// TIA Portal V20 export
FUNCTION_BLOCK "EmOverviewHomeCondition"   // FB5, LAD
// stored: MemoryReserve 100, SetENOAutomatically false
   VAR
      statMaxPageCount : Array[0..13] of Int;
      statPulse { ExternalAccessible := 'False'; ExternalVisible := 'False'; ExternalWritable := 'False'} : Array[0..199] of Bool;
      statLampOff { ExternalAccessible := 'False'; ExternalVisible := 'False'; ExternalWritable := 'False'} : Array[0..13] of Bool;
      statLampControl { ExternalAccessible := 'False'; ExternalVisible := 'False'; ExternalWritable := 'False'} : Bool;
   END_VAR
   VAR CONSTANT
      TRUE : Bool := TRUE;
      FALSE : Bool := FALSE;
   END_VAR
   VAR_TEMP   // added for the SCL form of the ladder/FBD networks
      _w1 : Bool;
      _w2 : Bool;
   END_VAR
BEGIN

REGION Network 1: Lamp Control
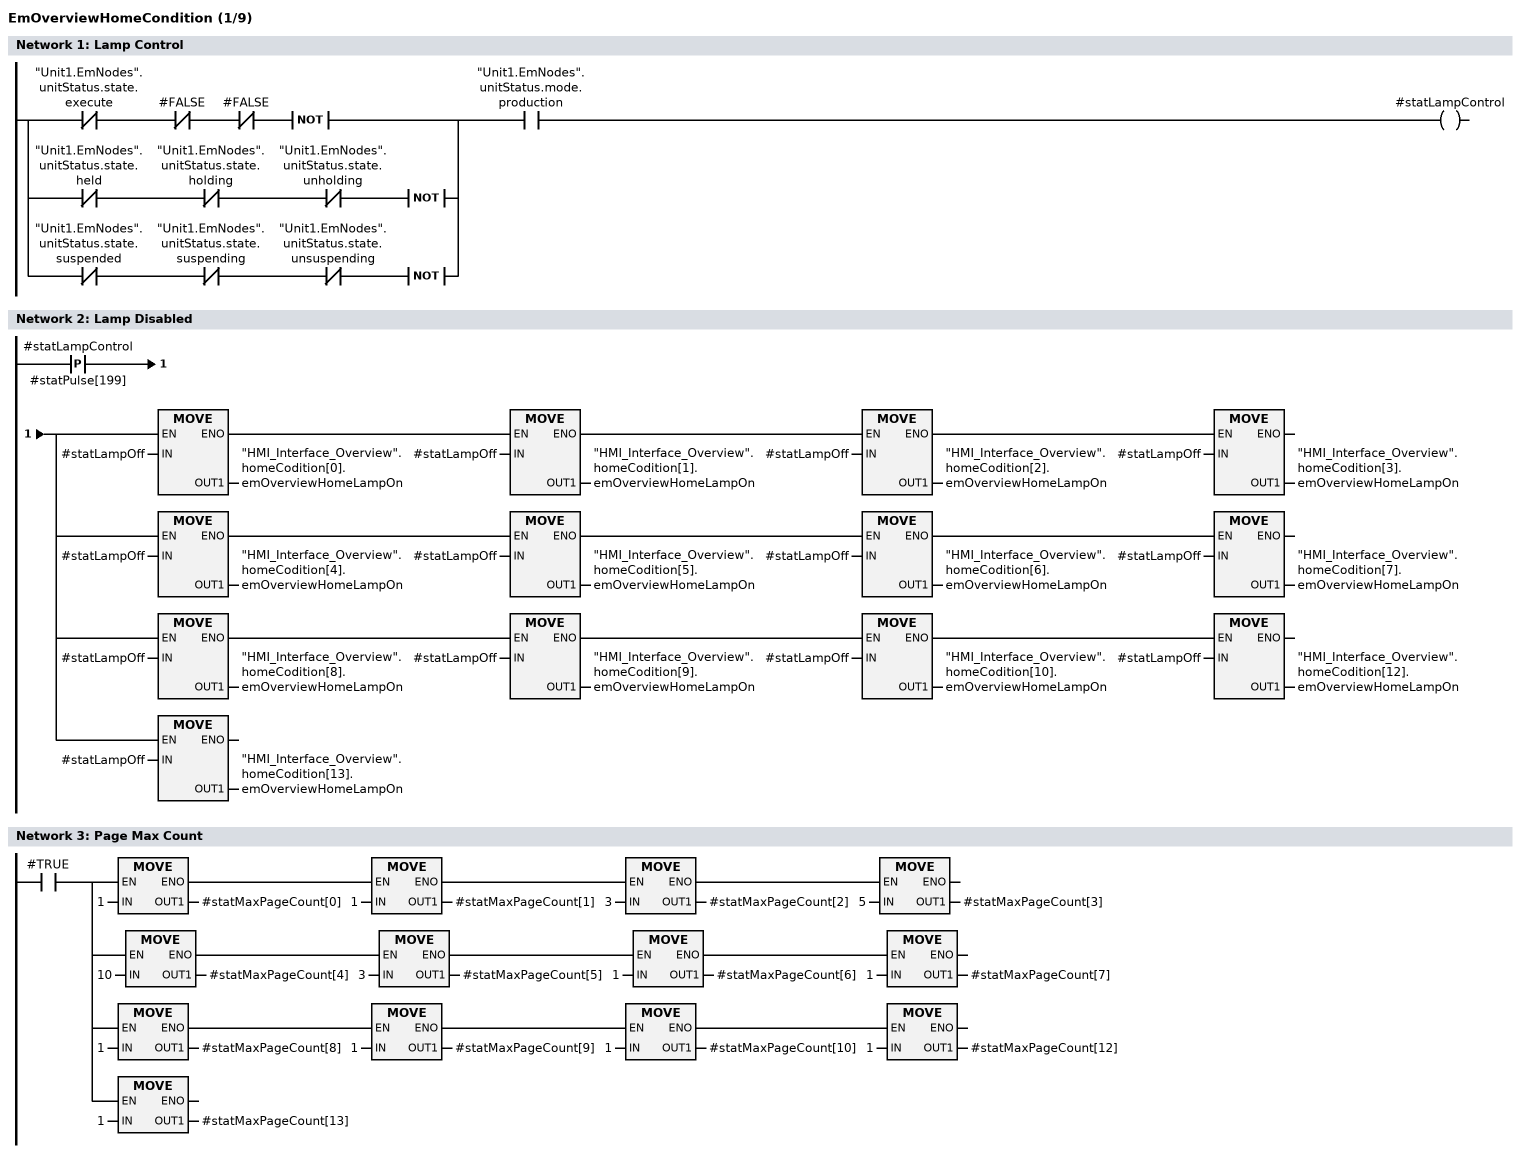
   RUNG wire#powerrail
      I_Contact( "Unit1.EmNodes".unitStatus.state.execute )
      I_Contact( #FALSE )
      I_Contact( #FALSE )
      Not()
      wire#w1
      Contact( "Unit1.EmNodes".unitStatus.mode.production )
      Coil( #statLampControl )
   END_RUNG
   RUNG wire#powerrail
      I_Contact( "Unit1.EmNodes".unitStatus.state.held )
      I_Contact( "Unit1.EmNodes".unitStatus.state.holding )
      I_Contact( "Unit1.EmNodes".unitStatus.state.unholding )
      Not()
   END_RUNG wire#w1
   RUNG wire#powerrail
      I_Contact( "Unit1.EmNodes".unitStatus.state.suspended )
      I_Contact( "Unit1.EmNodes".unitStatus.state.suspending )
      I_Contact( "Unit1.EmNodes".unitStatus.state.unsuspending )
      Not()
   END_RUNG wire#w1
   // the same network as SCL:
   #statLampControl := (NOT (NOT "Unit1.EmNodes".unitStatus.state.execute AND NOT #FALSE AND NOT #FALSE) OR NOT (NOT "Unit1.EmNodes".unitStatus.state.held AND NOT "Unit1.EmNodes".unitStatus.state.holding AND NOT "Unit1.EmNodes".unitStatus.state.unholding) OR NOT (NOT "Unit1.EmNodes".unitStatus.state.suspended AND NOT "Unit1.EmNodes".unitStatus.state.suspending AND NOT "Unit1.EmNodes".unitStatus.state.unsuspending)) AND "Unit1.EmNodes".unitStatus.mode.production;
END_REGION

REGION Network 2: Lamp Disabled
   RUNG wire#powerrail
      P_Contact(operand := #statLampControl, bit := #statPulse[199])
      wire#w1
      Move(in := #statLampOff, out1 => "HMI_Interface_Overview".homeCodition[0].emOverviewHomeLampOn)
      Move(in := #statLampOff, out1 => "HMI_Interface_Overview".homeCodition[1].emOverviewHomeLampOn)
      Move(in := #statLampOff, out1 => "HMI_Interface_Overview".homeCodition[2].emOverviewHomeLampOn)
      Move(in := #statLampOff, out1 => "HMI_Interface_Overview".homeCodition[3].emOverviewHomeLampOn)
   END_RUNG
   RUNG wire#w1
      Move(in := #statLampOff, out1 => "HMI_Interface_Overview".homeCodition[4].emOverviewHomeLampOn)
      Move(in := #statLampOff, out1 => "HMI_Interface_Overview".homeCodition[5].emOverviewHomeLampOn)
      Move(in := #statLampOff, out1 => "HMI_Interface_Overview".homeCodition[6].emOverviewHomeLampOn)
      Move(in := #statLampOff, out1 => "HMI_Interface_Overview".homeCodition[7].emOverviewHomeLampOn)
   END_RUNG
   RUNG wire#w1
      Move(in := #statLampOff, out1 => "HMI_Interface_Overview".homeCodition[8].emOverviewHomeLampOn)
      Move(in := #statLampOff, out1 => "HMI_Interface_Overview".homeCodition[9].emOverviewHomeLampOn)
      Move(in := #statLampOff, out1 => "HMI_Interface_Overview".homeCodition[10].emOverviewHomeLampOn)
      Move(in := #statLampOff, out1 => "HMI_Interface_Overview".homeCodition[12].emOverviewHomeLampOn)
   END_RUNG
   RUNG wire#w1
      Move(in := #statLampOff, out1 => "HMI_Interface_Overview".homeCodition[13].emOverviewHomeLampOn)
   END_RUNG
   // the same network as SCL:
   #_w1 := #statLampControl AND NOT #statPulse[199];   // rising edge of #statLampControl
   #statPulse[199] := #statLampControl;
   IF #_w1 THEN
       "HMI_Interface_Overview".homeCodition[0].emOverviewHomeLampOn := #statLampOff;
       "HMI_Interface_Overview".homeCodition[1].emOverviewHomeLampOn := #statLampOff;
       "HMI_Interface_Overview".homeCodition[2].emOverviewHomeLampOn := #statLampOff;
       "HMI_Interface_Overview".homeCodition[3].emOverviewHomeLampOn := #statLampOff;
       "HMI_Interface_Overview".homeCodition[4].emOverviewHomeLampOn := #statLampOff;
       "HMI_Interface_Overview".homeCodition[5].emOverviewHomeLampOn := #statLampOff;
       "HMI_Interface_Overview".homeCodition[6].emOverviewHomeLampOn := #statLampOff;
       "HMI_Interface_Overview".homeCodition[7].emOverviewHomeLampOn := #statLampOff;
       "HMI_Interface_Overview".homeCodition[8].emOverviewHomeLampOn := #statLampOff;
       "HMI_Interface_Overview".homeCodition[9].emOverviewHomeLampOn := #statLampOff;
       "HMI_Interface_Overview".homeCodition[10].emOverviewHomeLampOn := #statLampOff;
       "HMI_Interface_Overview".homeCodition[12].emOverviewHomeLampOn := #statLampOff;
       "HMI_Interface_Overview".homeCodition[13].emOverviewHomeLampOn := #statLampOff;
   END_IF;
END_REGION

REGION Network 3: Page Max Count
   RUNG wire#powerrail
      Contact( #TRUE )
      wire#w1
      Move(in := 1, out1 => #statMaxPageCount[0])
      Move(in := 1, out1 => #statMaxPageCount[1])
      Move(in := 3, out1 => #statMaxPageCount[2])
      Move(in := 5, out1 => #statMaxPageCount[3])
   END_RUNG
   RUNG wire#w1
      Move(in := 10, out1 => #statMaxPageCount[4])
      Move(in := 3, out1 => #statMaxPageCount[5])
      Move(in := 1, out1 => #statMaxPageCount[6])
      Move(in := 1, out1 => #statMaxPageCount[7])
   END_RUNG
   RUNG wire#w1
      Move(in := 1, out1 => #statMaxPageCount[8])
      Move(in := 1, out1 => #statMaxPageCount[9])
      Move(in := 1, out1 => #statMaxPageCount[10])
      Move(in := 1, out1 => #statMaxPageCount[12])
   END_RUNG
   RUNG wire#w1
      Move(in := 1, out1 => #statMaxPageCount[13])
   END_RUNG
   // the same network as SCL:
   IF #TRUE THEN
       #statMaxPageCount[0] := 1;
       #statMaxPageCount[1] := 1;
       #statMaxPageCount[2] := 3;
       #statMaxPageCount[3] := 5;
       #statMaxPageCount[4] := 10;
       #statMaxPageCount[5] := 3;
       #statMaxPageCount[6] := 1;
       #statMaxPageCount[7] := 1;
       #statMaxPageCount[8] := 1;
       #statMaxPageCount[9] := 1;
       #statMaxPageCount[10] := 1;
       #statMaxPageCount[12] := 1;
       #statMaxPageCount[13] := 1;
   END_IF;
END_REGION

REGION Network 4: Em 0 Page Index Control
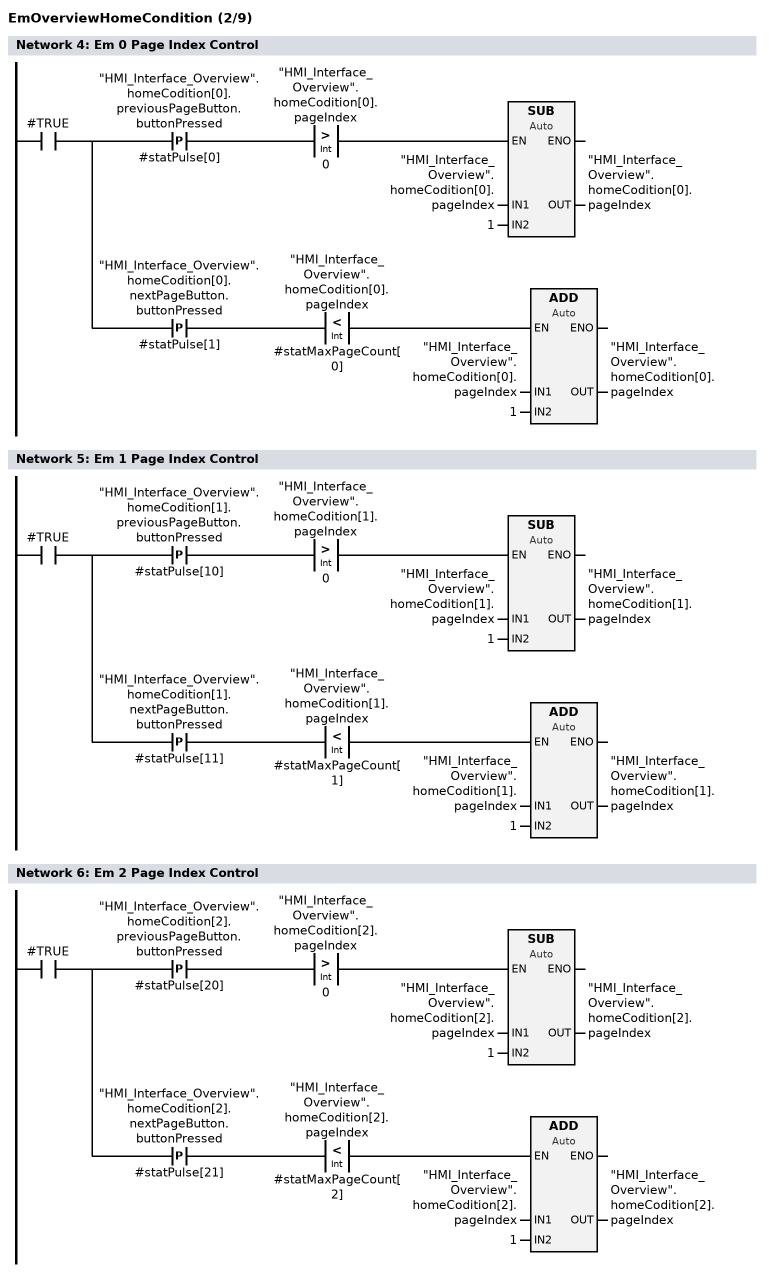
   RUNG wire#powerrail
      Contact( #TRUE )
      wire#w1
      P_Contact(operand := "HMI_Interface_Overview".homeCodition[0].previousPageButton.buttonPressed, bit := #statPulse[0])
      { S7_Templates := "SrcType := Int" } GT_Contact(in1 := "HMI_Interface_Overview".homeCodition[0].pageIndex, in2 := 0)
      Sub(in1 := "HMI_Interface_Overview".homeCodition[0].pageIndex, in2 := 1, out => "HMI_Interface_Overview".homeCodition[0].pageIndex)
   END_RUNG
   RUNG wire#w1
      P_Contact(operand := "HMI_Interface_Overview".homeCodition[0].nextPageButton.buttonPressed, bit := #statPulse[1])
      { S7_Templates := "SrcType := Int" } LT_Contact(in1 := "HMI_Interface_Overview".homeCodition[0].pageIndex, in2 := #statMaxPageCount[0])
      Add(in1 := "HMI_Interface_Overview".homeCodition[0].pageIndex, in2 := 1, out => "HMI_Interface_Overview".homeCodition[0].pageIndex)
   END_RUNG
   // the same network as SCL:
   #_w1 := #TRUE AND "HMI_Interface_Overview".homeCodition[0].previousPageButton.buttonPressed AND NOT #statPulse[0];   // rising edge of "HMI_Interface_Overview".homeCodition[0].previousPageButton.buttonPressed
   #statPulse[0] := "HMI_Interface_Overview".homeCodition[0].previousPageButton.buttonPressed;
   IF #_w1 AND ("HMI_Interface_Overview".homeCodition[0].pageIndex > 0) THEN
       "HMI_Interface_Overview".homeCodition[0].pageIndex := "HMI_Interface_Overview".homeCodition[0].pageIndex - 1;
   END_IF;
   #_w2 := #TRUE AND "HMI_Interface_Overview".homeCodition[0].nextPageButton.buttonPressed AND NOT #statPulse[1];   // rising edge of "HMI_Interface_Overview".homeCodition[0].nextPageButton.buttonPressed
   #statPulse[1] := "HMI_Interface_Overview".homeCodition[0].nextPageButton.buttonPressed;
   IF #_w2 AND ("HMI_Interface_Overview".homeCodition[0].pageIndex < #statMaxPageCount[0]) THEN
       "HMI_Interface_Overview".homeCodition[0].pageIndex := "HMI_Interface_Overview".homeCodition[0].pageIndex + 1;
   END_IF;
END_REGION

REGION Network 5: Em 1 Page Index Control
   RUNG wire#powerrail
      Contact( #TRUE )
      wire#w1
      P_Contact(operand := "HMI_Interface_Overview".homeCodition[1].previousPageButton.buttonPressed, bit := #statPulse[10])
      { S7_Templates := "SrcType := Int" } GT_Contact(in1 := "HMI_Interface_Overview".homeCodition[1].pageIndex, in2 := 0)
      Sub(in1 := "HMI_Interface_Overview".homeCodition[1].pageIndex, in2 := 1, out => "HMI_Interface_Overview".homeCodition[1].pageIndex)
   END_RUNG
   RUNG wire#w1
      P_Contact(operand := "HMI_Interface_Overview".homeCodition[1].nextPageButton.buttonPressed, bit := #statPulse[11])
      { S7_Templates := "SrcType := Int" } LT_Contact(in1 := "HMI_Interface_Overview".homeCodition[1].pageIndex, in2 := #statMaxPageCount[1])
      Add(in1 := "HMI_Interface_Overview".homeCodition[1].pageIndex, in2 := 1, out => "HMI_Interface_Overview".homeCodition[1].pageIndex)
   END_RUNG
   // the same network as SCL:
   #_w1 := #TRUE AND "HMI_Interface_Overview".homeCodition[1].previousPageButton.buttonPressed AND NOT #statPulse[10];   // rising edge of "HMI_Interface_Overview".homeCodition[1].previousPageButton.buttonPressed
   #statPulse[10] := "HMI_Interface_Overview".homeCodition[1].previousPageButton.buttonPressed;
   IF #_w1 AND ("HMI_Interface_Overview".homeCodition[1].pageIndex > 0) THEN
       "HMI_Interface_Overview".homeCodition[1].pageIndex := "HMI_Interface_Overview".homeCodition[1].pageIndex - 1;
   END_IF;
   #_w2 := #TRUE AND "HMI_Interface_Overview".homeCodition[1].nextPageButton.buttonPressed AND NOT #statPulse[11];   // rising edge of "HMI_Interface_Overview".homeCodition[1].nextPageButton.buttonPressed
   #statPulse[11] := "HMI_Interface_Overview".homeCodition[1].nextPageButton.buttonPressed;
   IF #_w2 AND ("HMI_Interface_Overview".homeCodition[1].pageIndex < #statMaxPageCount[1]) THEN
       "HMI_Interface_Overview".homeCodition[1].pageIndex := "HMI_Interface_Overview".homeCodition[1].pageIndex + 1;
   END_IF;
END_REGION

REGION Network 6: Em 2 Page Index Control
   RUNG wire#powerrail
      Contact( #TRUE )
      wire#w1
      P_Contact(operand := "HMI_Interface_Overview".homeCodition[2].previousPageButton.buttonPressed, bit := #statPulse[20])
      { S7_Templates := "SrcType := Int" } GT_Contact(in1 := "HMI_Interface_Overview".homeCodition[2].pageIndex, in2 := 0)
      Sub(in1 := "HMI_Interface_Overview".homeCodition[2].pageIndex, in2 := 1, out => "HMI_Interface_Overview".homeCodition[2].pageIndex)
   END_RUNG
   RUNG wire#w1
      P_Contact(operand := "HMI_Interface_Overview".homeCodition[2].nextPageButton.buttonPressed, bit := #statPulse[21])
      { S7_Templates := "SrcType := Int" } LT_Contact(in1 := "HMI_Interface_Overview".homeCodition[2].pageIndex, in2 := #statMaxPageCount[2])
      Add(in1 := "HMI_Interface_Overview".homeCodition[2].pageIndex, in2 := 1, out => "HMI_Interface_Overview".homeCodition[2].pageIndex)
   END_RUNG
   // the same network as SCL:
   #_w1 := #TRUE AND "HMI_Interface_Overview".homeCodition[2].previousPageButton.buttonPressed AND NOT #statPulse[20];   // rising edge of "HMI_Interface_Overview".homeCodition[2].previousPageButton.buttonPressed
   #statPulse[20] := "HMI_Interface_Overview".homeCodition[2].previousPageButton.buttonPressed;
   IF #_w1 AND ("HMI_Interface_Overview".homeCodition[2].pageIndex > 0) THEN
       "HMI_Interface_Overview".homeCodition[2].pageIndex := "HMI_Interface_Overview".homeCodition[2].pageIndex - 1;
   END_IF;
   #_w2 := #TRUE AND "HMI_Interface_Overview".homeCodition[2].nextPageButton.buttonPressed AND NOT #statPulse[21];   // rising edge of "HMI_Interface_Overview".homeCodition[2].nextPageButton.buttonPressed
   #statPulse[21] := "HMI_Interface_Overview".homeCodition[2].nextPageButton.buttonPressed;
   IF #_w2 AND ("HMI_Interface_Overview".homeCodition[2].pageIndex < #statMaxPageCount[2]) THEN
       "HMI_Interface_Overview".homeCodition[2].pageIndex := "HMI_Interface_Overview".homeCodition[2].pageIndex + 1;
   END_IF;
END_REGION

REGION Network 7: Em 3 Page Index Control
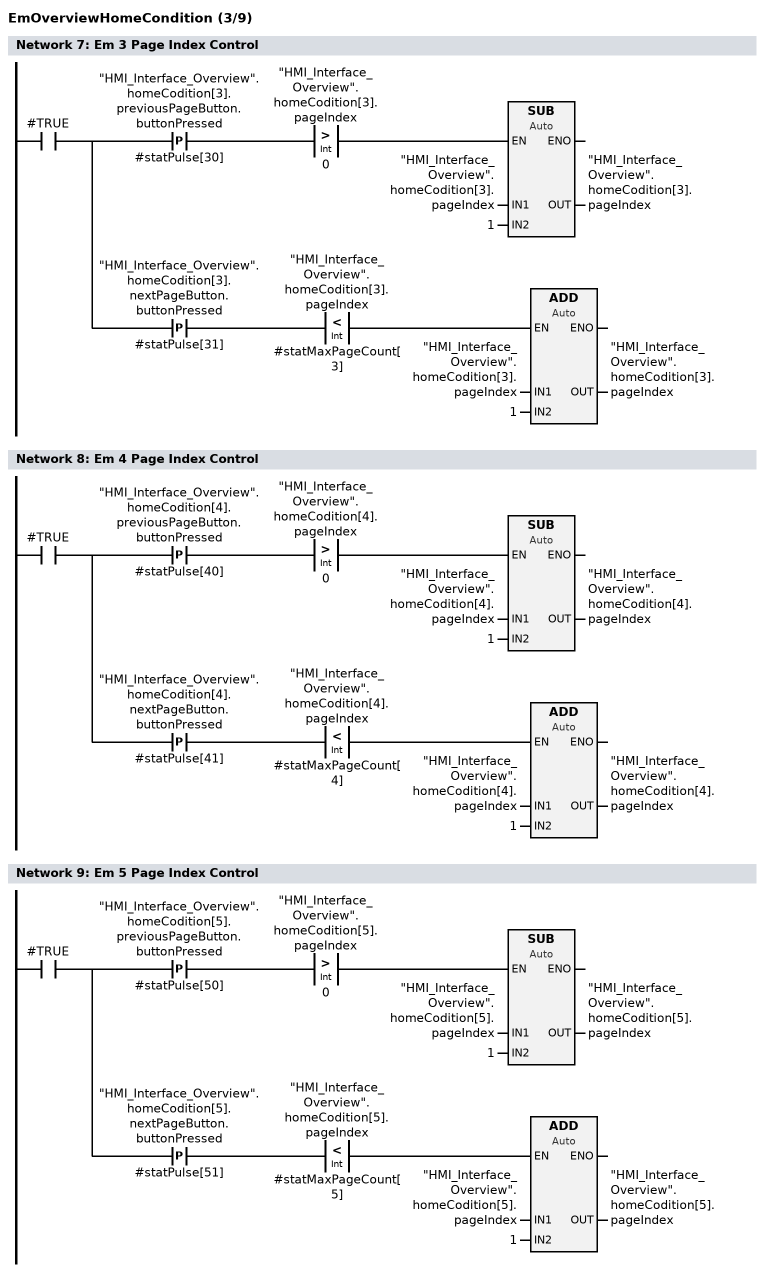
   RUNG wire#powerrail
      Contact( #TRUE )
      wire#w1
      P_Contact(operand := "HMI_Interface_Overview".homeCodition[3].previousPageButton.buttonPressed, bit := #statPulse[30])
      { S7_Templates := "SrcType := Int" } GT_Contact(in1 := "HMI_Interface_Overview".homeCodition[3].pageIndex, in2 := 0)
      Sub(in1 := "HMI_Interface_Overview".homeCodition[3].pageIndex, in2 := 1, out => "HMI_Interface_Overview".homeCodition[3].pageIndex)
   END_RUNG
   RUNG wire#w1
      P_Contact(operand := "HMI_Interface_Overview".homeCodition[3].nextPageButton.buttonPressed, bit := #statPulse[31])
      { S7_Templates := "SrcType := Int" } LT_Contact(in1 := "HMI_Interface_Overview".homeCodition[3].pageIndex, in2 := #statMaxPageCount[3])
      Add(in1 := "HMI_Interface_Overview".homeCodition[3].pageIndex, in2 := 1, out => "HMI_Interface_Overview".homeCodition[3].pageIndex)
   END_RUNG
   // the same network as SCL:
   #_w1 := #TRUE AND "HMI_Interface_Overview".homeCodition[3].previousPageButton.buttonPressed AND NOT #statPulse[30];   // rising edge of "HMI_Interface_Overview".homeCodition[3].previousPageButton.buttonPressed
   #statPulse[30] := "HMI_Interface_Overview".homeCodition[3].previousPageButton.buttonPressed;
   IF #_w1 AND ("HMI_Interface_Overview".homeCodition[3].pageIndex > 0) THEN
       "HMI_Interface_Overview".homeCodition[3].pageIndex := "HMI_Interface_Overview".homeCodition[3].pageIndex - 1;
   END_IF;
   #_w2 := #TRUE AND "HMI_Interface_Overview".homeCodition[3].nextPageButton.buttonPressed AND NOT #statPulse[31];   // rising edge of "HMI_Interface_Overview".homeCodition[3].nextPageButton.buttonPressed
   #statPulse[31] := "HMI_Interface_Overview".homeCodition[3].nextPageButton.buttonPressed;
   IF #_w2 AND ("HMI_Interface_Overview".homeCodition[3].pageIndex < #statMaxPageCount[3]) THEN
       "HMI_Interface_Overview".homeCodition[3].pageIndex := "HMI_Interface_Overview".homeCodition[3].pageIndex + 1;
   END_IF;
END_REGION

REGION Network 8: Em 4 Page Index Control
   RUNG wire#powerrail
      Contact( #TRUE )
      wire#w1
      P_Contact(operand := "HMI_Interface_Overview".homeCodition[4].previousPageButton.buttonPressed, bit := #statPulse[40])
      { S7_Templates := "SrcType := Int" } GT_Contact(in1 := "HMI_Interface_Overview".homeCodition[4].pageIndex, in2 := 0)
      Sub(in1 := "HMI_Interface_Overview".homeCodition[4].pageIndex, in2 := 1, out => "HMI_Interface_Overview".homeCodition[4].pageIndex)
   END_RUNG
   RUNG wire#w1
      P_Contact(operand := "HMI_Interface_Overview".homeCodition[4].nextPageButton.buttonPressed, bit := #statPulse[41])
      { S7_Templates := "SrcType := Int" } LT_Contact(in1 := "HMI_Interface_Overview".homeCodition[4].pageIndex, in2 := #statMaxPageCount[4])
      Add(in1 := "HMI_Interface_Overview".homeCodition[4].pageIndex, in2 := 1, out => "HMI_Interface_Overview".homeCodition[4].pageIndex)
   END_RUNG
   // the same network as SCL:
   #_w1 := #TRUE AND "HMI_Interface_Overview".homeCodition[4].previousPageButton.buttonPressed AND NOT #statPulse[40];   // rising edge of "HMI_Interface_Overview".homeCodition[4].previousPageButton.buttonPressed
   #statPulse[40] := "HMI_Interface_Overview".homeCodition[4].previousPageButton.buttonPressed;
   IF #_w1 AND ("HMI_Interface_Overview".homeCodition[4].pageIndex > 0) THEN
       "HMI_Interface_Overview".homeCodition[4].pageIndex := "HMI_Interface_Overview".homeCodition[4].pageIndex - 1;
   END_IF;
   #_w2 := #TRUE AND "HMI_Interface_Overview".homeCodition[4].nextPageButton.buttonPressed AND NOT #statPulse[41];   // rising edge of "HMI_Interface_Overview".homeCodition[4].nextPageButton.buttonPressed
   #statPulse[41] := "HMI_Interface_Overview".homeCodition[4].nextPageButton.buttonPressed;
   IF #_w2 AND ("HMI_Interface_Overview".homeCodition[4].pageIndex < #statMaxPageCount[4]) THEN
       "HMI_Interface_Overview".homeCodition[4].pageIndex := "HMI_Interface_Overview".homeCodition[4].pageIndex + 1;
   END_IF;
END_REGION

REGION Network 9: Em 5 Page Index Control
   RUNG wire#powerrail
      Contact( #TRUE )
      wire#w1
      P_Contact(operand := "HMI_Interface_Overview".homeCodition[5].previousPageButton.buttonPressed, bit := #statPulse[50])
      { S7_Templates := "SrcType := Int" } GT_Contact(in1 := "HMI_Interface_Overview".homeCodition[5].pageIndex, in2 := 0)
      Sub(in1 := "HMI_Interface_Overview".homeCodition[5].pageIndex, in2 := 1, out => "HMI_Interface_Overview".homeCodition[5].pageIndex)
   END_RUNG
   RUNG wire#w1
      P_Contact(operand := "HMI_Interface_Overview".homeCodition[5].nextPageButton.buttonPressed, bit := #statPulse[51])
      { S7_Templates := "SrcType := Int" } LT_Contact(in1 := "HMI_Interface_Overview".homeCodition[5].pageIndex, in2 := #statMaxPageCount[5])
      Add(in1 := "HMI_Interface_Overview".homeCodition[5].pageIndex, in2 := 1, out => "HMI_Interface_Overview".homeCodition[5].pageIndex)
   END_RUNG
   // the same network as SCL:
   #_w1 := #TRUE AND "HMI_Interface_Overview".homeCodition[5].previousPageButton.buttonPressed AND NOT #statPulse[50];   // rising edge of "HMI_Interface_Overview".homeCodition[5].previousPageButton.buttonPressed
   #statPulse[50] := "HMI_Interface_Overview".homeCodition[5].previousPageButton.buttonPressed;
   IF #_w1 AND ("HMI_Interface_Overview".homeCodition[5].pageIndex > 0) THEN
       "HMI_Interface_Overview".homeCodition[5].pageIndex := "HMI_Interface_Overview".homeCodition[5].pageIndex - 1;
   END_IF;
   #_w2 := #TRUE AND "HMI_Interface_Overview".homeCodition[5].nextPageButton.buttonPressed AND NOT #statPulse[51];   // rising edge of "HMI_Interface_Overview".homeCodition[5].nextPageButton.buttonPressed
   #statPulse[51] := "HMI_Interface_Overview".homeCodition[5].nextPageButton.buttonPressed;
   IF #_w2 AND ("HMI_Interface_Overview".homeCodition[5].pageIndex < #statMaxPageCount[5]) THEN
       "HMI_Interface_Overview".homeCodition[5].pageIndex := "HMI_Interface_Overview".homeCodition[5].pageIndex + 1;
   END_IF;
END_REGION

REGION Network 10: Em 6 Page Index Control
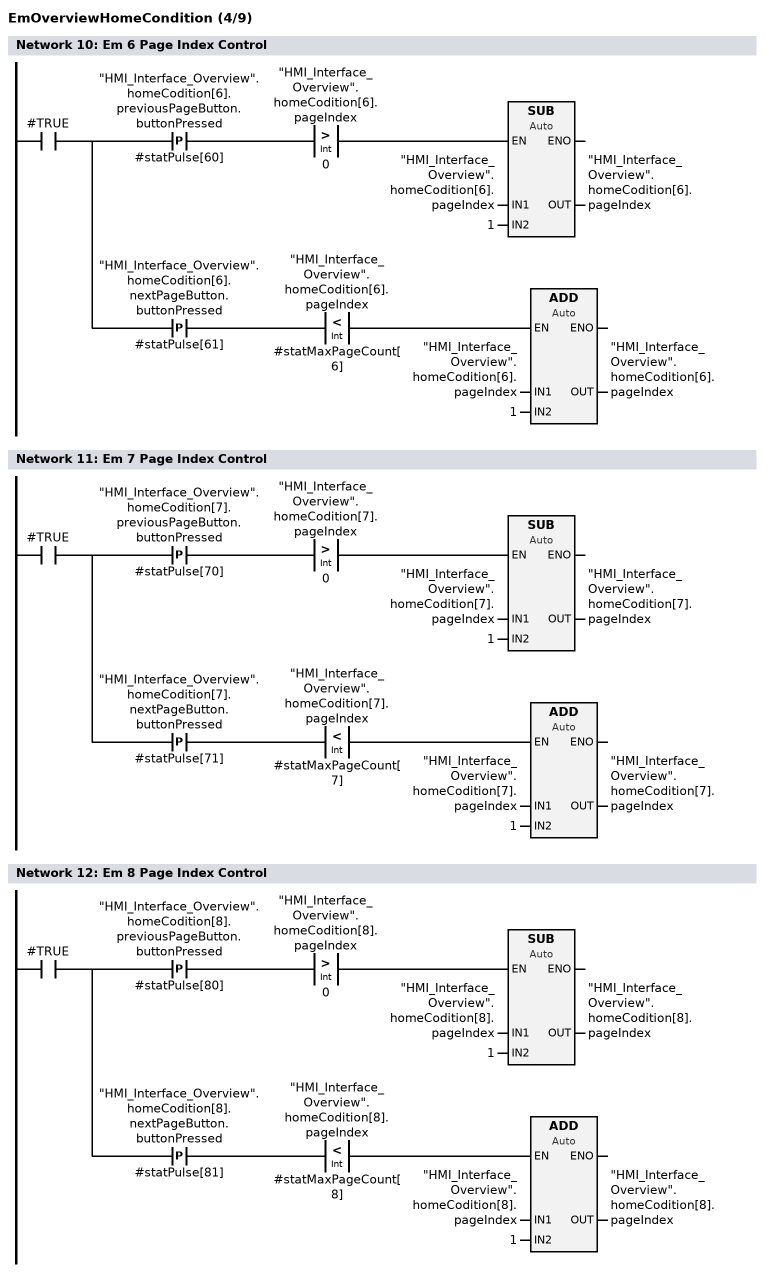
   RUNG wire#powerrail
      Contact( #TRUE )
      wire#w1
      P_Contact(operand := "HMI_Interface_Overview".homeCodition[6].previousPageButton.buttonPressed, bit := #statPulse[60])
      { S7_Templates := "SrcType := Int" } GT_Contact(in1 := "HMI_Interface_Overview".homeCodition[6].pageIndex, in2 := 0)
      Sub(in1 := "HMI_Interface_Overview".homeCodition[6].pageIndex, in2 := 1, out => "HMI_Interface_Overview".homeCodition[6].pageIndex)
   END_RUNG
   RUNG wire#w1
      P_Contact(operand := "HMI_Interface_Overview".homeCodition[6].nextPageButton.buttonPressed, bit := #statPulse[61])
      { S7_Templates := "SrcType := Int" } LT_Contact(in1 := "HMI_Interface_Overview".homeCodition[6].pageIndex, in2 := #statMaxPageCount[6])
      Add(in1 := "HMI_Interface_Overview".homeCodition[6].pageIndex, in2 := 1, out => "HMI_Interface_Overview".homeCodition[6].pageIndex)
   END_RUNG
   // the same network as SCL:
   #_w1 := #TRUE AND "HMI_Interface_Overview".homeCodition[6].previousPageButton.buttonPressed AND NOT #statPulse[60];   // rising edge of "HMI_Interface_Overview".homeCodition[6].previousPageButton.buttonPressed
   #statPulse[60] := "HMI_Interface_Overview".homeCodition[6].previousPageButton.buttonPressed;
   IF #_w1 AND ("HMI_Interface_Overview".homeCodition[6].pageIndex > 0) THEN
       "HMI_Interface_Overview".homeCodition[6].pageIndex := "HMI_Interface_Overview".homeCodition[6].pageIndex - 1;
   END_IF;
   #_w2 := #TRUE AND "HMI_Interface_Overview".homeCodition[6].nextPageButton.buttonPressed AND NOT #statPulse[61];   // rising edge of "HMI_Interface_Overview".homeCodition[6].nextPageButton.buttonPressed
   #statPulse[61] := "HMI_Interface_Overview".homeCodition[6].nextPageButton.buttonPressed;
   IF #_w2 AND ("HMI_Interface_Overview".homeCodition[6].pageIndex < #statMaxPageCount[6]) THEN
       "HMI_Interface_Overview".homeCodition[6].pageIndex := "HMI_Interface_Overview".homeCodition[6].pageIndex + 1;
   END_IF;
END_REGION

REGION Network 11: Em 7 Page Index Control
   RUNG wire#powerrail
      Contact( #TRUE )
      wire#w1
      P_Contact(operand := "HMI_Interface_Overview".homeCodition[7].previousPageButton.buttonPressed, bit := #statPulse[70])
      { S7_Templates := "SrcType := Int" } GT_Contact(in1 := "HMI_Interface_Overview".homeCodition[7].pageIndex, in2 := 0)
      Sub(in1 := "HMI_Interface_Overview".homeCodition[7].pageIndex, in2 := 1, out => "HMI_Interface_Overview".homeCodition[7].pageIndex)
   END_RUNG
   RUNG wire#w1
      P_Contact(operand := "HMI_Interface_Overview".homeCodition[7].nextPageButton.buttonPressed, bit := #statPulse[71])
      { S7_Templates := "SrcType := Int" } LT_Contact(in1 := "HMI_Interface_Overview".homeCodition[7].pageIndex, in2 := #statMaxPageCount[7])
      Add(in1 := "HMI_Interface_Overview".homeCodition[7].pageIndex, in2 := 1, out => "HMI_Interface_Overview".homeCodition[7].pageIndex)
   END_RUNG
   // the same network as SCL:
   #_w1 := #TRUE AND "HMI_Interface_Overview".homeCodition[7].previousPageButton.buttonPressed AND NOT #statPulse[70];   // rising edge of "HMI_Interface_Overview".homeCodition[7].previousPageButton.buttonPressed
   #statPulse[70] := "HMI_Interface_Overview".homeCodition[7].previousPageButton.buttonPressed;
   IF #_w1 AND ("HMI_Interface_Overview".homeCodition[7].pageIndex > 0) THEN
       "HMI_Interface_Overview".homeCodition[7].pageIndex := "HMI_Interface_Overview".homeCodition[7].pageIndex - 1;
   END_IF;
   #_w2 := #TRUE AND "HMI_Interface_Overview".homeCodition[7].nextPageButton.buttonPressed AND NOT #statPulse[71];   // rising edge of "HMI_Interface_Overview".homeCodition[7].nextPageButton.buttonPressed
   #statPulse[71] := "HMI_Interface_Overview".homeCodition[7].nextPageButton.buttonPressed;
   IF #_w2 AND ("HMI_Interface_Overview".homeCodition[7].pageIndex < #statMaxPageCount[7]) THEN
       "HMI_Interface_Overview".homeCodition[7].pageIndex := "HMI_Interface_Overview".homeCodition[7].pageIndex + 1;
   END_IF;
END_REGION

REGION Network 12: Em 8 Page Index Control
   RUNG wire#powerrail
      Contact( #TRUE )
      wire#w1
      P_Contact(operand := "HMI_Interface_Overview".homeCodition[8].previousPageButton.buttonPressed, bit := #statPulse[80])
      { S7_Templates := "SrcType := Int" } GT_Contact(in1 := "HMI_Interface_Overview".homeCodition[8].pageIndex, in2 := 0)
      Sub(in1 := "HMI_Interface_Overview".homeCodition[8].pageIndex, in2 := 1, out => "HMI_Interface_Overview".homeCodition[8].pageIndex)
   END_RUNG
   RUNG wire#w1
      P_Contact(operand := "HMI_Interface_Overview".homeCodition[8].nextPageButton.buttonPressed, bit := #statPulse[81])
      { S7_Templates := "SrcType := Int" } LT_Contact(in1 := "HMI_Interface_Overview".homeCodition[8].pageIndex, in2 := #statMaxPageCount[8])
      Add(in1 := "HMI_Interface_Overview".homeCodition[8].pageIndex, in2 := 1, out => "HMI_Interface_Overview".homeCodition[8].pageIndex)
   END_RUNG
   // the same network as SCL:
   #_w1 := #TRUE AND "HMI_Interface_Overview".homeCodition[8].previousPageButton.buttonPressed AND NOT #statPulse[80];   // rising edge of "HMI_Interface_Overview".homeCodition[8].previousPageButton.buttonPressed
   #statPulse[80] := "HMI_Interface_Overview".homeCodition[8].previousPageButton.buttonPressed;
   IF #_w1 AND ("HMI_Interface_Overview".homeCodition[8].pageIndex > 0) THEN
       "HMI_Interface_Overview".homeCodition[8].pageIndex := "HMI_Interface_Overview".homeCodition[8].pageIndex - 1;
   END_IF;
   #_w2 := #TRUE AND "HMI_Interface_Overview".homeCodition[8].nextPageButton.buttonPressed AND NOT #statPulse[81];   // rising edge of "HMI_Interface_Overview".homeCodition[8].nextPageButton.buttonPressed
   #statPulse[81] := "HMI_Interface_Overview".homeCodition[8].nextPageButton.buttonPressed;
   IF #_w2 AND ("HMI_Interface_Overview".homeCodition[8].pageIndex < #statMaxPageCount[8]) THEN
       "HMI_Interface_Overview".homeCodition[8].pageIndex := "HMI_Interface_Overview".homeCodition[8].pageIndex + 1;
   END_IF;
END_REGION

REGION Network 13: Em 9 Page Index Control
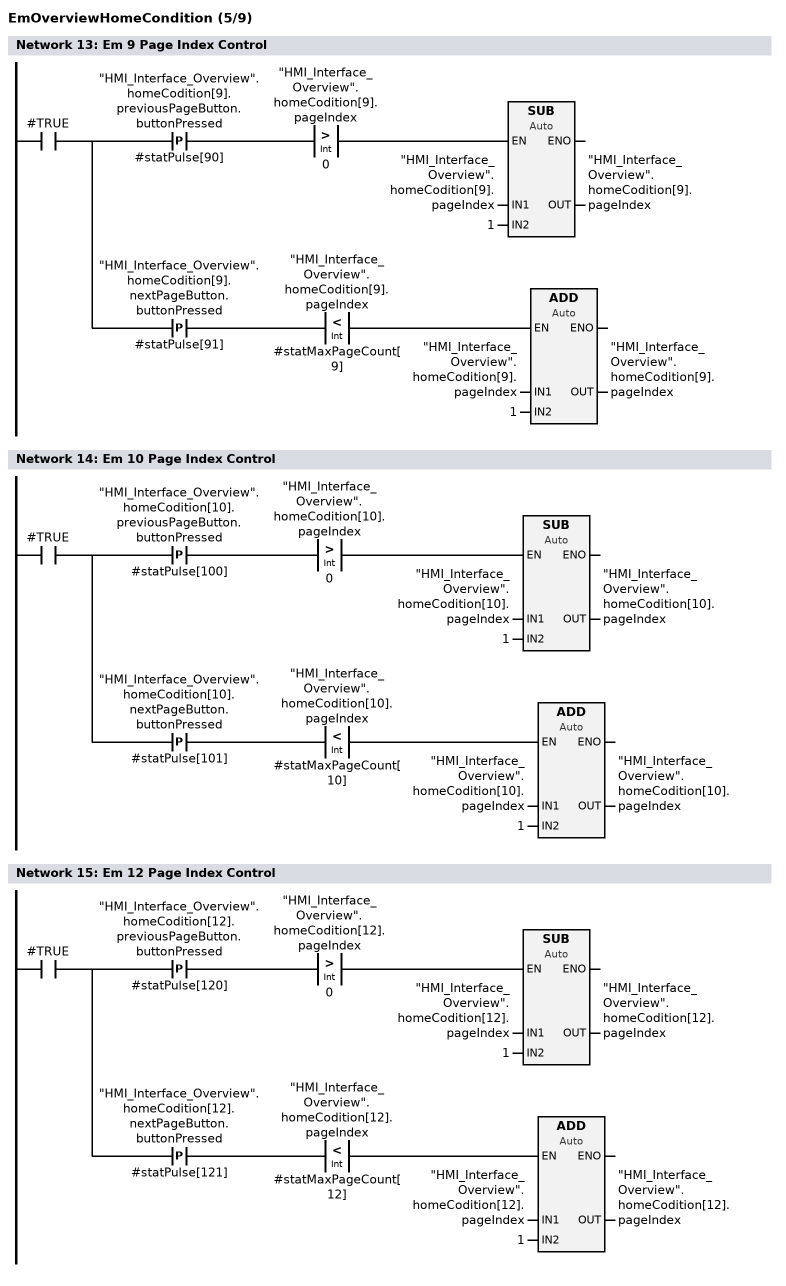
   RUNG wire#powerrail
      Contact( #TRUE )
      wire#w1
      P_Contact(operand := "HMI_Interface_Overview".homeCodition[9].previousPageButton.buttonPressed, bit := #statPulse[90])
      { S7_Templates := "SrcType := Int" } GT_Contact(in1 := "HMI_Interface_Overview".homeCodition[9].pageIndex, in2 := 0)
      Sub(in1 := "HMI_Interface_Overview".homeCodition[9].pageIndex, in2 := 1, out => "HMI_Interface_Overview".homeCodition[9].pageIndex)
   END_RUNG
   RUNG wire#w1
      P_Contact(operand := "HMI_Interface_Overview".homeCodition[9].nextPageButton.buttonPressed, bit := #statPulse[91])
      { S7_Templates := "SrcType := Int" } LT_Contact(in1 := "HMI_Interface_Overview".homeCodition[9].pageIndex, in2 := #statMaxPageCount[9])
      Add(in1 := "HMI_Interface_Overview".homeCodition[9].pageIndex, in2 := 1, out => "HMI_Interface_Overview".homeCodition[9].pageIndex)
   END_RUNG
   // the same network as SCL:
   #_w1 := #TRUE AND "HMI_Interface_Overview".homeCodition[9].previousPageButton.buttonPressed AND NOT #statPulse[90];   // rising edge of "HMI_Interface_Overview".homeCodition[9].previousPageButton.buttonPressed
   #statPulse[90] := "HMI_Interface_Overview".homeCodition[9].previousPageButton.buttonPressed;
   IF #_w1 AND ("HMI_Interface_Overview".homeCodition[9].pageIndex > 0) THEN
       "HMI_Interface_Overview".homeCodition[9].pageIndex := "HMI_Interface_Overview".homeCodition[9].pageIndex - 1;
   END_IF;
   #_w2 := #TRUE AND "HMI_Interface_Overview".homeCodition[9].nextPageButton.buttonPressed AND NOT #statPulse[91];   // rising edge of "HMI_Interface_Overview".homeCodition[9].nextPageButton.buttonPressed
   #statPulse[91] := "HMI_Interface_Overview".homeCodition[9].nextPageButton.buttonPressed;
   IF #_w2 AND ("HMI_Interface_Overview".homeCodition[9].pageIndex < #statMaxPageCount[9]) THEN
       "HMI_Interface_Overview".homeCodition[9].pageIndex := "HMI_Interface_Overview".homeCodition[9].pageIndex + 1;
   END_IF;
END_REGION

REGION Network 14: Em 10 Page Index Control
   RUNG wire#powerrail
      Contact( #TRUE )
      wire#w1
      P_Contact(operand := "HMI_Interface_Overview".homeCodition[10].previousPageButton.buttonPressed, bit := #statPulse[100])
      { S7_Templates := "SrcType := Int" } GT_Contact(in1 := "HMI_Interface_Overview".homeCodition[10].pageIndex, in2 := 0)
      Sub(in1 := "HMI_Interface_Overview".homeCodition[10].pageIndex, in2 := 1, out => "HMI_Interface_Overview".homeCodition[10].pageIndex)
   END_RUNG
   RUNG wire#w1
      P_Contact(operand := "HMI_Interface_Overview".homeCodition[10].nextPageButton.buttonPressed, bit := #statPulse[101])
      { S7_Templates := "SrcType := Int" } LT_Contact(in1 := "HMI_Interface_Overview".homeCodition[10].pageIndex, in2 := #statMaxPageCount[10])
      Add(in1 := "HMI_Interface_Overview".homeCodition[10].pageIndex, in2 := 1, out => "HMI_Interface_Overview".homeCodition[10].pageIndex)
   END_RUNG
   // the same network as SCL:
   #_w1 := #TRUE AND "HMI_Interface_Overview".homeCodition[10].previousPageButton.buttonPressed AND NOT #statPulse[100];   // rising edge of "HMI_Interface_Overview".homeCodition[10].previousPageButton.buttonPressed
   #statPulse[100] := "HMI_Interface_Overview".homeCodition[10].previousPageButton.buttonPressed;
   IF #_w1 AND ("HMI_Interface_Overview".homeCodition[10].pageIndex > 0) THEN
       "HMI_Interface_Overview".homeCodition[10].pageIndex := "HMI_Interface_Overview".homeCodition[10].pageIndex - 1;
   END_IF;
   #_w2 := #TRUE AND "HMI_Interface_Overview".homeCodition[10].nextPageButton.buttonPressed AND NOT #statPulse[101];   // rising edge of "HMI_Interface_Overview".homeCodition[10].nextPageButton.buttonPressed
   #statPulse[101] := "HMI_Interface_Overview".homeCodition[10].nextPageButton.buttonPressed;
   IF #_w2 AND ("HMI_Interface_Overview".homeCodition[10].pageIndex < #statMaxPageCount[10]) THEN
       "HMI_Interface_Overview".homeCodition[10].pageIndex := "HMI_Interface_Overview".homeCodition[10].pageIndex + 1;
   END_IF;
END_REGION

REGION Network 15: Em 12 Page Index Control
   RUNG wire#powerrail
      Contact( #TRUE )
      wire#w1
      P_Contact(operand := "HMI_Interface_Overview".homeCodition[12].previousPageButton.buttonPressed, bit := #statPulse[120])
      { S7_Templates := "SrcType := Int" } GT_Contact(in1 := "HMI_Interface_Overview".homeCodition[12].pageIndex, in2 := 0)
      Sub(in1 := "HMI_Interface_Overview".homeCodition[12].pageIndex, in2 := 1, out => "HMI_Interface_Overview".homeCodition[12].pageIndex)
   END_RUNG
   RUNG wire#w1
      P_Contact(operand := "HMI_Interface_Overview".homeCodition[12].nextPageButton.buttonPressed, bit := #statPulse[121])
      { S7_Templates := "SrcType := Int" } LT_Contact(in1 := "HMI_Interface_Overview".homeCodition[12].pageIndex, in2 := #statMaxPageCount[12])
      Add(in1 := "HMI_Interface_Overview".homeCodition[12].pageIndex, in2 := 1, out => "HMI_Interface_Overview".homeCodition[12].pageIndex)
   END_RUNG
   // the same network as SCL:
   #_w1 := #TRUE AND "HMI_Interface_Overview".homeCodition[12].previousPageButton.buttonPressed AND NOT #statPulse[120];   // rising edge of "HMI_Interface_Overview".homeCodition[12].previousPageButton.buttonPressed
   #statPulse[120] := "HMI_Interface_Overview".homeCodition[12].previousPageButton.buttonPressed;
   IF #_w1 AND ("HMI_Interface_Overview".homeCodition[12].pageIndex > 0) THEN
       "HMI_Interface_Overview".homeCodition[12].pageIndex := "HMI_Interface_Overview".homeCodition[12].pageIndex - 1;
   END_IF;
   #_w2 := #TRUE AND "HMI_Interface_Overview".homeCodition[12].nextPageButton.buttonPressed AND NOT #statPulse[121];   // rising edge of "HMI_Interface_Overview".homeCodition[12].nextPageButton.buttonPressed
   #statPulse[121] := "HMI_Interface_Overview".homeCodition[12].nextPageButton.buttonPressed;
   IF #_w2 AND ("HMI_Interface_Overview".homeCodition[12].pageIndex < #statMaxPageCount[12]) THEN
       "HMI_Interface_Overview".homeCodition[12].pageIndex := "HMI_Interface_Overview".homeCodition[12].pageIndex + 1;
   END_IF;
END_REGION

REGION Network 16: Em 13 Page Index Control
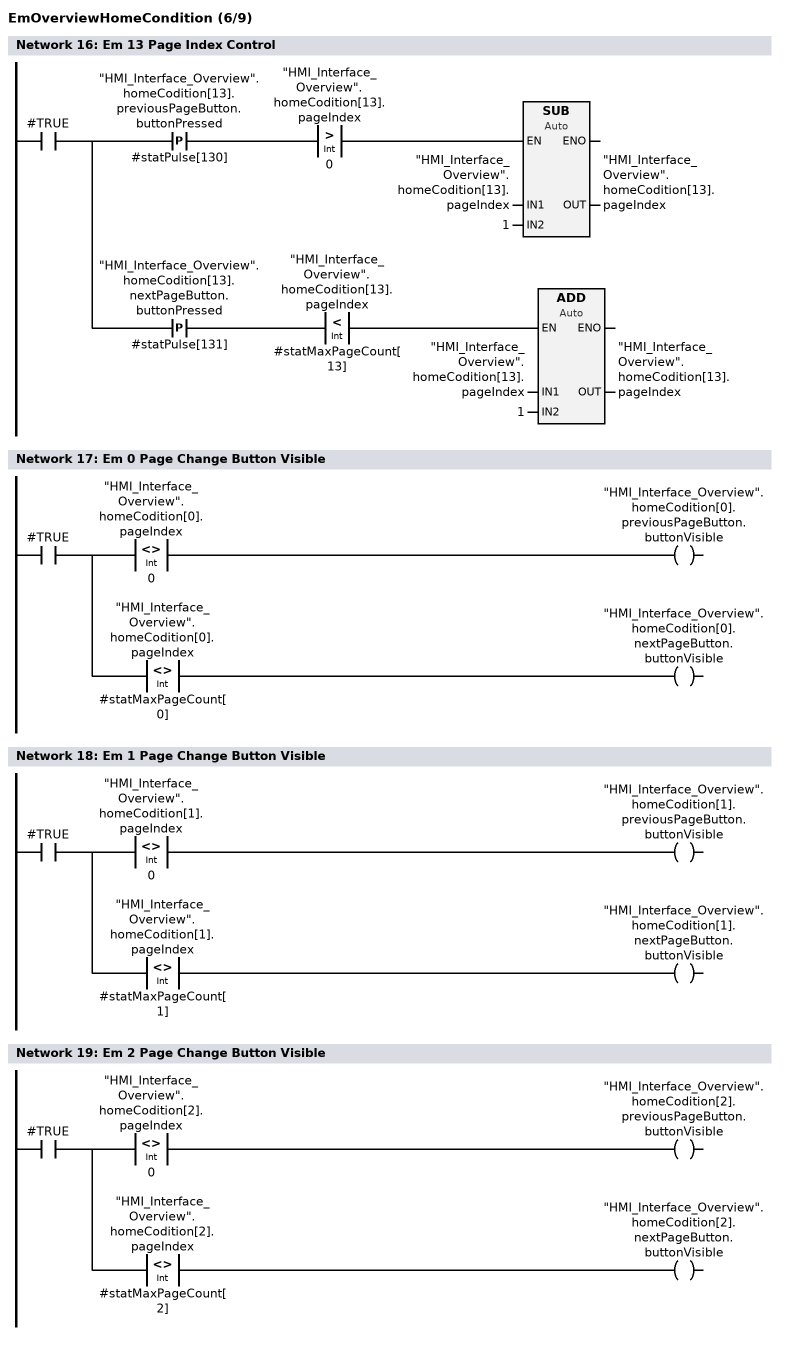
   RUNG wire#powerrail
      Contact( #TRUE )
      wire#w1
      P_Contact(operand := "HMI_Interface_Overview".homeCodition[13].previousPageButton.buttonPressed, bit := #statPulse[130])
      { S7_Templates := "SrcType := Int" } GT_Contact(in1 := "HMI_Interface_Overview".homeCodition[13].pageIndex, in2 := 0)
      Sub(in1 := "HMI_Interface_Overview".homeCodition[13].pageIndex, in2 := 1, out => "HMI_Interface_Overview".homeCodition[13].pageIndex)
   END_RUNG
   RUNG wire#w1
      P_Contact(operand := "HMI_Interface_Overview".homeCodition[13].nextPageButton.buttonPressed, bit := #statPulse[131])
      { S7_Templates := "SrcType := Int" } LT_Contact(in1 := "HMI_Interface_Overview".homeCodition[13].pageIndex, in2 := #statMaxPageCount[13])
      Add(in1 := "HMI_Interface_Overview".homeCodition[13].pageIndex, in2 := 1, out => "HMI_Interface_Overview".homeCodition[13].pageIndex)
   END_RUNG
   // the same network as SCL:
   #_w1 := #TRUE AND "HMI_Interface_Overview".homeCodition[13].previousPageButton.buttonPressed AND NOT #statPulse[130];   // rising edge of "HMI_Interface_Overview".homeCodition[13].previousPageButton.buttonPressed
   #statPulse[130] := "HMI_Interface_Overview".homeCodition[13].previousPageButton.buttonPressed;
   IF #_w1 AND ("HMI_Interface_Overview".homeCodition[13].pageIndex > 0) THEN
       "HMI_Interface_Overview".homeCodition[13].pageIndex := "HMI_Interface_Overview".homeCodition[13].pageIndex - 1;
   END_IF;
   #_w2 := #TRUE AND "HMI_Interface_Overview".homeCodition[13].nextPageButton.buttonPressed AND NOT #statPulse[131];   // rising edge of "HMI_Interface_Overview".homeCodition[13].nextPageButton.buttonPressed
   #statPulse[131] := "HMI_Interface_Overview".homeCodition[13].nextPageButton.buttonPressed;
   IF #_w2 AND ("HMI_Interface_Overview".homeCodition[13].pageIndex < #statMaxPageCount[13]) THEN
       "HMI_Interface_Overview".homeCodition[13].pageIndex := "HMI_Interface_Overview".homeCodition[13].pageIndex + 1;
   END_IF;
END_REGION

REGION Network 17: Em 0 Page Change Button Visible
   RUNG wire#powerrail
      Contact( #TRUE )
      wire#w1
      { S7_Templates := "SrcType := Int" } NE_Contact(in1 := "HMI_Interface_Overview".homeCodition[0].pageIndex, in2 := 0)
      Coil( "HMI_Interface_Overview".homeCodition[0].previousPageButton.buttonVisible )
   END_RUNG
   RUNG wire#w1
      { S7_Templates := "SrcType := Int" } NE_Contact(in1 := "HMI_Interface_Overview".homeCodition[0].pageIndex, in2 := #statMaxPageCount[0])
      Coil( "HMI_Interface_Overview".homeCodition[0].nextPageButton.buttonVisible )
   END_RUNG
   // the same network as SCL:
   "HMI_Interface_Overview".homeCodition[0].previousPageButton.buttonVisible := #TRUE AND ("HMI_Interface_Overview".homeCodition[0].pageIndex <> 0);
   "HMI_Interface_Overview".homeCodition[0].nextPageButton.buttonVisible := #TRUE AND ("HMI_Interface_Overview".homeCodition[0].pageIndex <> #statMaxPageCount[0]);
END_REGION

REGION Network 18: Em 1 Page Change Button Visible
   RUNG wire#powerrail
      Contact( #TRUE )
      wire#w1
      { S7_Templates := "SrcType := Int" } NE_Contact(in1 := "HMI_Interface_Overview".homeCodition[1].pageIndex, in2 := 0)
      Coil( "HMI_Interface_Overview".homeCodition[1].previousPageButton.buttonVisible )
   END_RUNG
   RUNG wire#w1
      { S7_Templates := "SrcType := Int" } NE_Contact(in1 := "HMI_Interface_Overview".homeCodition[1].pageIndex, in2 := #statMaxPageCount[1])
      Coil( "HMI_Interface_Overview".homeCodition[1].nextPageButton.buttonVisible )
   END_RUNG
   // the same network as SCL:
   "HMI_Interface_Overview".homeCodition[1].previousPageButton.buttonVisible := #TRUE AND ("HMI_Interface_Overview".homeCodition[1].pageIndex <> 0);
   "HMI_Interface_Overview".homeCodition[1].nextPageButton.buttonVisible := #TRUE AND ("HMI_Interface_Overview".homeCodition[1].pageIndex <> #statMaxPageCount[1]);
END_REGION

REGION Network 19: Em 2 Page Change Button Visible
   RUNG wire#powerrail
      Contact( #TRUE )
      wire#w1
      { S7_Templates := "SrcType := Int" } NE_Contact(in1 := "HMI_Interface_Overview".homeCodition[2].pageIndex, in2 := 0)
      Coil( "HMI_Interface_Overview".homeCodition[2].previousPageButton.buttonVisible )
   END_RUNG
   RUNG wire#w1
      { S7_Templates := "SrcType := Int" } NE_Contact(in1 := "HMI_Interface_Overview".homeCodition[2].pageIndex, in2 := #statMaxPageCount[2])
      Coil( "HMI_Interface_Overview".homeCodition[2].nextPageButton.buttonVisible )
   END_RUNG
   // the same network as SCL:
   "HMI_Interface_Overview".homeCodition[2].previousPageButton.buttonVisible := #TRUE AND ("HMI_Interface_Overview".homeCodition[2].pageIndex <> 0);
   "HMI_Interface_Overview".homeCodition[2].nextPageButton.buttonVisible := #TRUE AND ("HMI_Interface_Overview".homeCodition[2].pageIndex <> #statMaxPageCount[2]);
END_REGION

REGION Network 20: Em 3 Page Change Button Visible
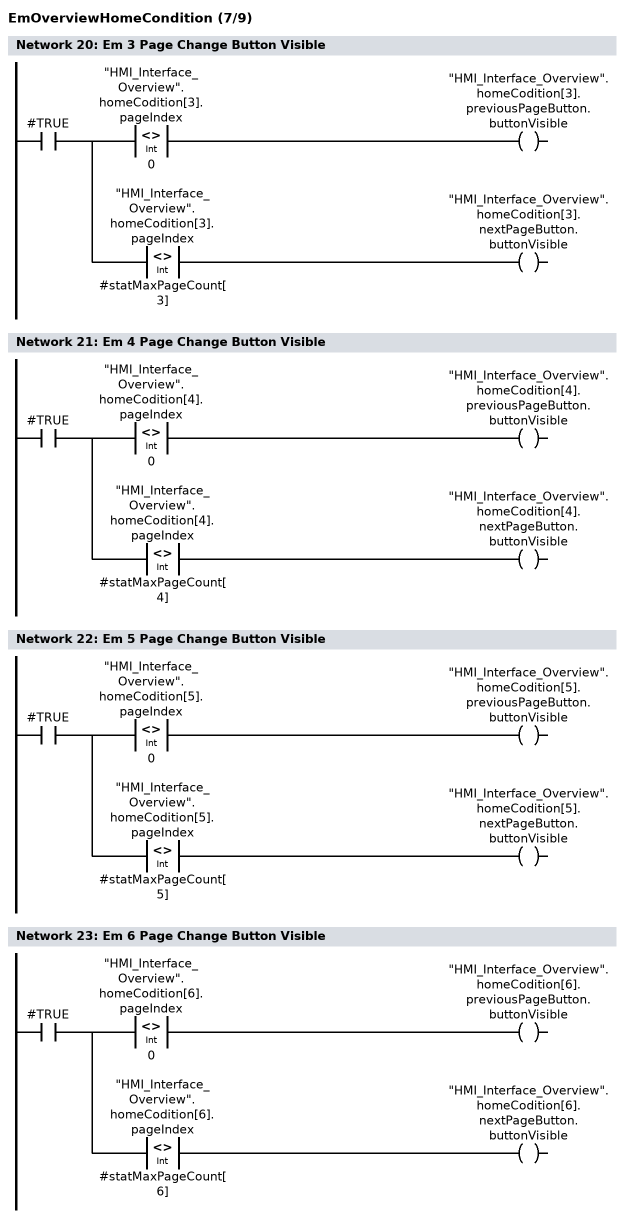
   RUNG wire#powerrail
      Contact( #TRUE )
      wire#w1
      { S7_Templates := "SrcType := Int" } NE_Contact(in1 := "HMI_Interface_Overview".homeCodition[3].pageIndex, in2 := 0)
      Coil( "HMI_Interface_Overview".homeCodition[3].previousPageButton.buttonVisible )
   END_RUNG
   RUNG wire#w1
      { S7_Templates := "SrcType := Int" } NE_Contact(in1 := "HMI_Interface_Overview".homeCodition[3].pageIndex, in2 := #statMaxPageCount[3])
      Coil( "HMI_Interface_Overview".homeCodition[3].nextPageButton.buttonVisible )
   END_RUNG
   // the same network as SCL:
   "HMI_Interface_Overview".homeCodition[3].previousPageButton.buttonVisible := #TRUE AND ("HMI_Interface_Overview".homeCodition[3].pageIndex <> 0);
   "HMI_Interface_Overview".homeCodition[3].nextPageButton.buttonVisible := #TRUE AND ("HMI_Interface_Overview".homeCodition[3].pageIndex <> #statMaxPageCount[3]);
END_REGION

REGION Network 21: Em 4 Page Change Button Visible
   RUNG wire#powerrail
      Contact( #TRUE )
      wire#w1
      { S7_Templates := "SrcType := Int" } NE_Contact(in1 := "HMI_Interface_Overview".homeCodition[4].pageIndex, in2 := 0)
      Coil( "HMI_Interface_Overview".homeCodition[4].previousPageButton.buttonVisible )
   END_RUNG
   RUNG wire#w1
      { S7_Templates := "SrcType := Int" } NE_Contact(in1 := "HMI_Interface_Overview".homeCodition[4].pageIndex, in2 := #statMaxPageCount[4])
      Coil( "HMI_Interface_Overview".homeCodition[4].nextPageButton.buttonVisible )
   END_RUNG
   // the same network as SCL:
   "HMI_Interface_Overview".homeCodition[4].previousPageButton.buttonVisible := #TRUE AND ("HMI_Interface_Overview".homeCodition[4].pageIndex <> 0);
   "HMI_Interface_Overview".homeCodition[4].nextPageButton.buttonVisible := #TRUE AND ("HMI_Interface_Overview".homeCodition[4].pageIndex <> #statMaxPageCount[4]);
END_REGION

REGION Network 22: Em 5 Page Change Button Visible
   RUNG wire#powerrail
      Contact( #TRUE )
      wire#w1
      { S7_Templates := "SrcType := Int" } NE_Contact(in1 := "HMI_Interface_Overview".homeCodition[5].pageIndex, in2 := 0)
      Coil( "HMI_Interface_Overview".homeCodition[5].previousPageButton.buttonVisible )
   END_RUNG
   RUNG wire#w1
      { S7_Templates := "SrcType := Int" } NE_Contact(in1 := "HMI_Interface_Overview".homeCodition[5].pageIndex, in2 := #statMaxPageCount[5])
      Coil( "HMI_Interface_Overview".homeCodition[5].nextPageButton.buttonVisible )
   END_RUNG
   // the same network as SCL:
   "HMI_Interface_Overview".homeCodition[5].previousPageButton.buttonVisible := #TRUE AND ("HMI_Interface_Overview".homeCodition[5].pageIndex <> 0);
   "HMI_Interface_Overview".homeCodition[5].nextPageButton.buttonVisible := #TRUE AND ("HMI_Interface_Overview".homeCodition[5].pageIndex <> #statMaxPageCount[5]);
END_REGION

REGION Network 23: Em 6 Page Change Button Visible
   RUNG wire#powerrail
      Contact( #TRUE )
      wire#w1
      { S7_Templates := "SrcType := Int" } NE_Contact(in1 := "HMI_Interface_Overview".homeCodition[6].pageIndex, in2 := 0)
      Coil( "HMI_Interface_Overview".homeCodition[6].previousPageButton.buttonVisible )
   END_RUNG
   RUNG wire#w1
      { S7_Templates := "SrcType := Int" } NE_Contact(in1 := "HMI_Interface_Overview".homeCodition[6].pageIndex, in2 := #statMaxPageCount[6])
      Coil( "HMI_Interface_Overview".homeCodition[6].nextPageButton.buttonVisible )
   END_RUNG
   // the same network as SCL:
   "HMI_Interface_Overview".homeCodition[6].previousPageButton.buttonVisible := #TRUE AND ("HMI_Interface_Overview".homeCodition[6].pageIndex <> 0);
   "HMI_Interface_Overview".homeCodition[6].nextPageButton.buttonVisible := #TRUE AND ("HMI_Interface_Overview".homeCodition[6].pageIndex <> #statMaxPageCount[6]);
END_REGION

REGION Network 24: Em 7 Page Change Button Visible
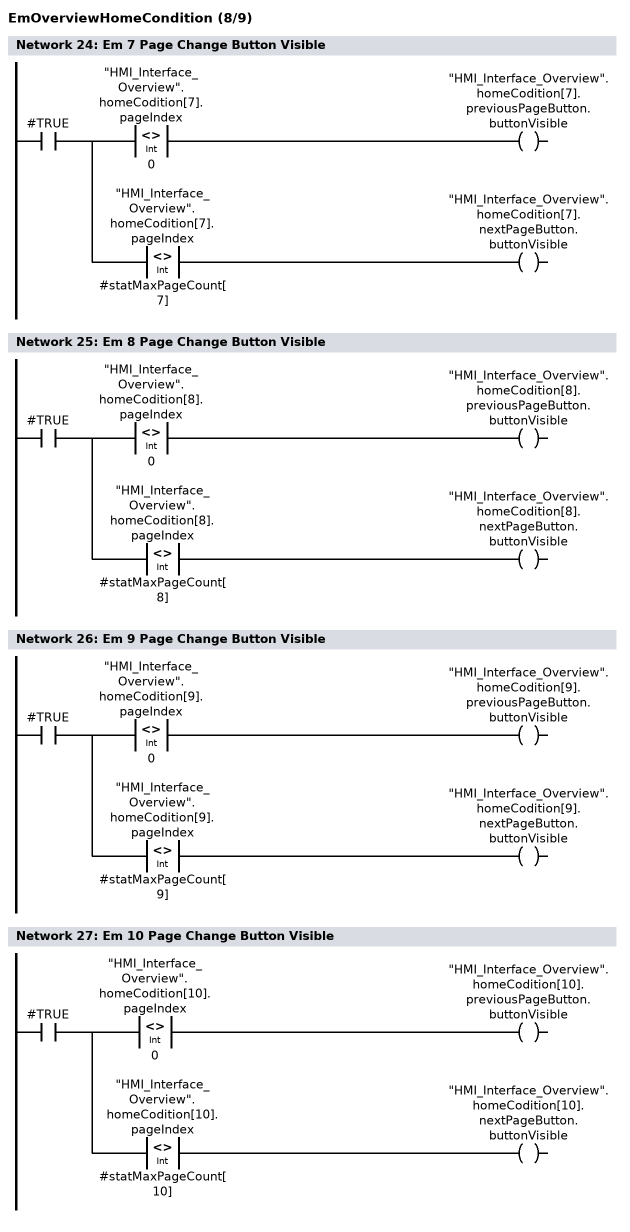
   RUNG wire#powerrail
      Contact( #TRUE )
      wire#w1
      { S7_Templates := "SrcType := Int" } NE_Contact(in1 := "HMI_Interface_Overview".homeCodition[7].pageIndex, in2 := 0)
      Coil( "HMI_Interface_Overview".homeCodition[7].previousPageButton.buttonVisible )
   END_RUNG
   RUNG wire#w1
      { S7_Templates := "SrcType := Int" } NE_Contact(in1 := "HMI_Interface_Overview".homeCodition[7].pageIndex, in2 := #statMaxPageCount[7])
      Coil( "HMI_Interface_Overview".homeCodition[7].nextPageButton.buttonVisible )
   END_RUNG
   // the same network as SCL:
   "HMI_Interface_Overview".homeCodition[7].previousPageButton.buttonVisible := #TRUE AND ("HMI_Interface_Overview".homeCodition[7].pageIndex <> 0);
   "HMI_Interface_Overview".homeCodition[7].nextPageButton.buttonVisible := #TRUE AND ("HMI_Interface_Overview".homeCodition[7].pageIndex <> #statMaxPageCount[7]);
END_REGION

REGION Network 25: Em 8 Page Change Button Visible
   RUNG wire#powerrail
      Contact( #TRUE )
      wire#w1
      { S7_Templates := "SrcType := Int" } NE_Contact(in1 := "HMI_Interface_Overview".homeCodition[8].pageIndex, in2 := 0)
      Coil( "HMI_Interface_Overview".homeCodition[8].previousPageButton.buttonVisible )
   END_RUNG
   RUNG wire#w1
      { S7_Templates := "SrcType := Int" } NE_Contact(in1 := "HMI_Interface_Overview".homeCodition[8].pageIndex, in2 := #statMaxPageCount[8])
      Coil( "HMI_Interface_Overview".homeCodition[8].nextPageButton.buttonVisible )
   END_RUNG
   // the same network as SCL:
   "HMI_Interface_Overview".homeCodition[8].previousPageButton.buttonVisible := #TRUE AND ("HMI_Interface_Overview".homeCodition[8].pageIndex <> 0);
   "HMI_Interface_Overview".homeCodition[8].nextPageButton.buttonVisible := #TRUE AND ("HMI_Interface_Overview".homeCodition[8].pageIndex <> #statMaxPageCount[8]);
END_REGION

REGION Network 26: Em 9 Page Change Button Visible
   RUNG wire#powerrail
      Contact( #TRUE )
      wire#w1
      { S7_Templates := "SrcType := Int" } NE_Contact(in1 := "HMI_Interface_Overview".homeCodition[9].pageIndex, in2 := 0)
      Coil( "HMI_Interface_Overview".homeCodition[9].previousPageButton.buttonVisible )
   END_RUNG
   RUNG wire#w1
      { S7_Templates := "SrcType := Int" } NE_Contact(in1 := "HMI_Interface_Overview".homeCodition[9].pageIndex, in2 := #statMaxPageCount[9])
      Coil( "HMI_Interface_Overview".homeCodition[9].nextPageButton.buttonVisible )
   END_RUNG
   // the same network as SCL:
   "HMI_Interface_Overview".homeCodition[9].previousPageButton.buttonVisible := #TRUE AND ("HMI_Interface_Overview".homeCodition[9].pageIndex <> 0);
   "HMI_Interface_Overview".homeCodition[9].nextPageButton.buttonVisible := #TRUE AND ("HMI_Interface_Overview".homeCodition[9].pageIndex <> #statMaxPageCount[9]);
END_REGION

REGION Network 27: Em 10 Page Change Button Visible
   RUNG wire#powerrail
      Contact( #TRUE )
      wire#w1
      { S7_Templates := "SrcType := Int" } NE_Contact(in1 := "HMI_Interface_Overview".homeCodition[10].pageIndex, in2 := 0)
      Coil( "HMI_Interface_Overview".homeCodition[10].previousPageButton.buttonVisible )
   END_RUNG
   RUNG wire#w1
      { S7_Templates := "SrcType := Int" } NE_Contact(in1 := "HMI_Interface_Overview".homeCodition[10].pageIndex, in2 := #statMaxPageCount[10])
      Coil( "HMI_Interface_Overview".homeCodition[10].nextPageButton.buttonVisible )
   END_RUNG
   // the same network as SCL:
   "HMI_Interface_Overview".homeCodition[10].previousPageButton.buttonVisible := #TRUE AND ("HMI_Interface_Overview".homeCodition[10].pageIndex <> 0);
   "HMI_Interface_Overview".homeCodition[10].nextPageButton.buttonVisible := #TRUE AND ("HMI_Interface_Overview".homeCodition[10].pageIndex <> #statMaxPageCount[10]);
END_REGION

REGION Network 28: Em 12 Page Change Button Visible
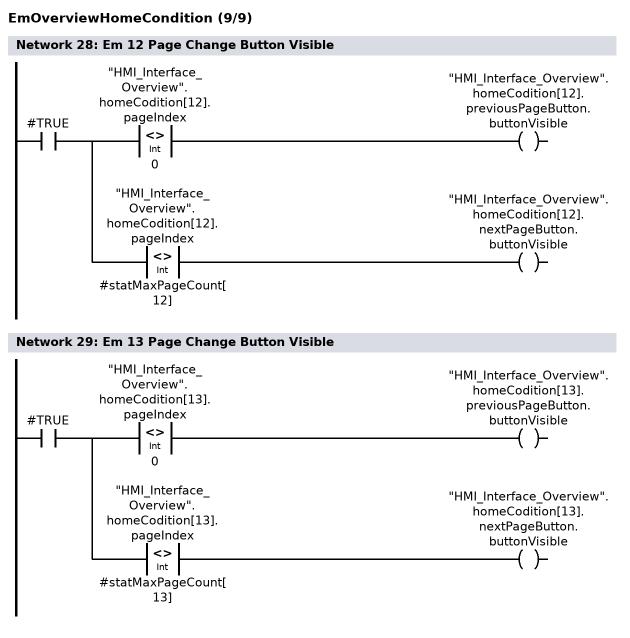
   RUNG wire#powerrail
      Contact( #TRUE )
      wire#w1
      { S7_Templates := "SrcType := Int" } NE_Contact(in1 := "HMI_Interface_Overview".homeCodition[12].pageIndex, in2 := 0)
      Coil( "HMI_Interface_Overview".homeCodition[12].previousPageButton.buttonVisible )
   END_RUNG
   RUNG wire#w1
      { S7_Templates := "SrcType := Int" } NE_Contact(in1 := "HMI_Interface_Overview".homeCodition[12].pageIndex, in2 := #statMaxPageCount[12])
      Coil( "HMI_Interface_Overview".homeCodition[12].nextPageButton.buttonVisible )
   END_RUNG
   // the same network as SCL:
   "HMI_Interface_Overview".homeCodition[12].previousPageButton.buttonVisible := #TRUE AND ("HMI_Interface_Overview".homeCodition[12].pageIndex <> 0);
   "HMI_Interface_Overview".homeCodition[12].nextPageButton.buttonVisible := #TRUE AND ("HMI_Interface_Overview".homeCodition[12].pageIndex <> #statMaxPageCount[12]);
END_REGION

REGION Network 29: Em 13 Page Change Button Visible
   RUNG wire#powerrail
      Contact( #TRUE )
      wire#w1
      { S7_Templates := "SrcType := Int" } NE_Contact(in1 := "HMI_Interface_Overview".homeCodition[13].pageIndex, in2 := 0)
      Coil( "HMI_Interface_Overview".homeCodition[13].previousPageButton.buttonVisible )
   END_RUNG
   RUNG wire#w1
      { S7_Templates := "SrcType := Int" } NE_Contact(in1 := "HMI_Interface_Overview".homeCodition[13].pageIndex, in2 := #statMaxPageCount[13])
      Coil( "HMI_Interface_Overview".homeCodition[13].nextPageButton.buttonVisible )
   END_RUNG
   // the same network as SCL:
   "HMI_Interface_Overview".homeCodition[13].previousPageButton.buttonVisible := #TRUE AND ("HMI_Interface_Overview".homeCodition[13].pageIndex <> 0);
   "HMI_Interface_Overview".homeCodition[13].nextPageButton.buttonVisible := #TRUE AND ("HMI_Interface_Overview".homeCodition[13].pageIndex <> #statMaxPageCount[13]);
END_REGION

REGION Network 30 (SCL): Em 0 Page Index Mapping
   REGION Page Index

       // Index 0
       IF "HMI_Interface_Overview".homeCodition[0].pageIndex = 0 THEN
           "HMI_Interface_Overview".homeCodition[0].emOverviewTitle := WSTRING#'Home Conidtion 0';
           "HMI_Interface_Overview".homeCodition[0].emOverviewCmName[0] := WSTRING#'Stacker 1 NG Box Loading';
           "HMI_Interface_Overview".homeCodition[0].emOverviewCmName[1] := WSTRING#'Stacker 1 NG Box Unit Mover';
           "HMI_Interface_Overview".homeCodition[0].emOverviewCmName[2] := WSTRING#'Stacker 1 NG Box Clamp Left';
           "HMI_Interface_Overview".homeCodition[0].emOverviewCmName[3] := WSTRING#'Stacker 1 NG Box Clamp Right';
           "HMI_Interface_Overview".homeCodition[0].emOverviewCmName[4] := WSTRING#'Stacker 1 NG Box Clamp Mover';
           "HMI_Interface_Overview".homeCodition[0].emOverviewCmName[5] := WSTRING#'Spare';
           "HMI_Interface_Overview".homeCodition[0].emOverviewCmName[6] := WSTRING#'Spare';
           "HMI_Interface_Overview".homeCodition[0].emOverviewCmName[7] := WSTRING#'Spare';
           "HMI_Interface_Overview".homeCodition[0].emOverviewCmName[8] := WSTRING#'Spare';
           "HMI_Interface_Overview".homeCodition[0].emOverviewCmName[9] := WSTRING#'Spare';
           "HMI_Interface_Overview".homeCodition[0].emOverviewCmName[10] := WSTRING#'Spare';
           "HMI_Interface_Overview".homeCodition[0].emOverviewCmName[11] := WSTRING#'Spare';
           "HMI_Interface_Overview".homeCodition[0].emOverviewCmName[12] := WSTRING#'Spare';
           "HMI_Interface_Overview".homeCodition[0].emOverviewCmName[13] := WSTRING#'Spare';
           "HMI_Interface_Overview".homeCodition[0].emOverviewCmPositionName[0] := WSTRING#'Up';
           "HMI_Interface_Overview".homeCodition[0].emOverviewCmPositionName[1] := WSTRING#'Backward';
           "HMI_Interface_Overview".homeCodition[0].emOverviewCmPositionName[2] := WSTRING#'Open';
           "HMI_Interface_Overview".homeCodition[0].emOverviewCmPositionName[3] := WSTRING#'Open';
           "HMI_Interface_Overview".homeCodition[0].emOverviewCmPositionName[4] := WSTRING#'Open';
           "HMI_Interface_Overview".homeCodition[0].emOverviewCmPositionName[5] := WSTRING#'Spare';
           "HMI_Interface_Overview".homeCodition[0].emOverviewCmPositionName[6] := WSTRING#'Spare';
           "HMI_Interface_Overview".homeCodition[0].emOverviewCmPositionName[7] := WSTRING#'Spare';
           "HMI_Interface_Overview".homeCodition[0].emOverviewCmPositionName[8] := WSTRING#'Spare';
           "HMI_Interface_Overview".homeCodition[0].emOverviewCmPositionName[9] := WSTRING#'Spare';
           "HMI_Interface_Overview".homeCodition[0].emOverviewCmPositionName[10] := WSTRING#'Spare';
           "HMI_Interface_Overview".homeCodition[0].emOverviewCmPositionName[11] := WSTRING#'Spare';
           "HMI_Interface_Overview".homeCodition[0].emOverviewCmPositionName[12] := WSTRING#'Spare';
           "HMI_Interface_Overview".homeCodition[0].emOverviewCmPositionName[13] := WSTRING#'Spare';
           IF NOT #statLampControl THEN
               "HMI_Interface_Overview".homeCodition[0].emOverviewHomeLampOn[0] := "Unit1.Em0.HmiInterface".cmStacker1NgBoxLoadingUpDown.monitoring.inHomePos;
               "HMI_Interface_Overview".homeCodition[0].emOverviewHomeLampOn[1] := "Unit1.Em0.HmiInterface".cmStacker1NgBoxUnitMoverBwdFwd.monitoring.inHomePos;
               "HMI_Interface_Overview".homeCodition[0].emOverviewHomeLampOn[2] := "Unit1.Em0.HmiInterface".cmStacker1NgBoxClampLeftOpenClose.monitoring.inHomePos;
               "HMI_Interface_Overview".homeCodition[0].emOverviewHomeLampOn[3] := "Unit1.Em0.HmiInterface".cmStacker1NgBoxClampRightOpenClose.monitoring.inHomePos;
               "HMI_Interface_Overview".homeCodition[0].emOverviewHomeLampOn[4] := "Unit1.Em0.HmiInterface".cmStacker1NgBoxClampMoverOpenClose.monitoring.inHomePos;
               "HMI_Interface_Overview".homeCodition[0].emOverviewHomeLampOn[5] := FALSE;
               "HMI_Interface_Overview".homeCodition[0].emOverviewHomeLampOn[6] := FALSE;
               "HMI_Interface_Overview".homeCodition[0].emOverviewHomeLampOn[7] := FALSE;
               "HMI_Interface_Overview".homeCodition[0].emOverviewHomeLampOn[8] := FALSE;
               "HMI_Interface_Overview".homeCodition[0].emOverviewHomeLampOn[9] := FALSE;
               "HMI_Interface_Overview".homeCodition[0].emOverviewHomeLampOn[10] := FALSE;
               "HMI_Interface_Overview".homeCodition[0].emOverviewHomeLampOn[11] := FALSE;
               "HMI_Interface_Overview".homeCodition[0].emOverviewHomeLampOn[12] := FALSE;
               "HMI_Interface_Overview".homeCodition[0].emOverviewHomeLampOn[13] := FALSE;
           END_IF;
       END_IF;

       // Index 1
       IF "HMI_Interface_Overview".homeCodition[0].pageIndex = 1 THEN
           "HMI_Interface_Overview".homeCodition[0].emOverviewTitle := WSTRING#'Home Conidtion 1';
           "HMI_Interface_Overview".homeCodition[0].emOverviewCmName[0] := WSTRING#'Stacker 1 NG Box Loading';
           "HMI_Interface_Overview".homeCodition[0].emOverviewCmName[1] := WSTRING#'Stacker 1 NG Box Unit Mover';
           "HMI_Interface_Overview".homeCodition[0].emOverviewCmName[2] := WSTRING#'Stacker 1 NG Box Clamp Left';
           "HMI_Interface_Overview".homeCodition[0].emOverviewCmName[3] := WSTRING#'Stacker 1 NG Box Clamp Right';
           "HMI_Interface_Overview".homeCodition[0].emOverviewCmName[4] := WSTRING#'Stacker 1 NG Box Clamp Mover';
           "HMI_Interface_Overview".homeCodition[0].emOverviewCmName[5] := WSTRING#'Spare';
           "HMI_Interface_Overview".homeCodition[0].emOverviewCmName[6] := WSTRING#'Spare';
           "HMI_Interface_Overview".homeCodition[0].emOverviewCmName[7] := WSTRING#'Spare';
           "HMI_Interface_Overview".homeCodition[0].emOverviewCmName[8] := WSTRING#'Spare';
           "HMI_Interface_Overview".homeCodition[0].emOverviewCmName[9] := WSTRING#'Spare';
           "HMI_Interface_Overview".homeCodition[0].emOverviewCmName[10] := WSTRING#'Spare';
           "HMI_Interface_Overview".homeCodition[0].emOverviewCmName[11] := WSTRING#'Spare';
           "HMI_Interface_Overview".homeCodition[0].emOverviewCmName[12] := WSTRING#'Spare';
           "HMI_Interface_Overview".homeCodition[0].emOverviewCmName[13] := WSTRING#'Spare';
           "HMI_Interface_Overview".homeCodition[0].emOverviewCmPositionName[0] := WSTRING#'Up';
           "HMI_Interface_Overview".homeCodition[0].emOverviewCmPositionName[1] := WSTRING#'Backward';
           "HMI_Interface_Overview".homeCodition[0].emOverviewCmPositionName[2] := WSTRING#'Close';
           "HMI_Interface_Overview".homeCodition[0].emOverviewCmPositionName[3] := WSTRING#'Close';
           "HMI_Interface_Overview".homeCodition[0].emOverviewCmPositionName[4] := WSTRING#'Close';
           "HMI_Interface_Overview".homeCodition[0].emOverviewCmPositionName[5] := WSTRING#'Spare';
           "HMI_Interface_Overview".homeCodition[0].emOverviewCmPositionName[6] := WSTRING#'Spare';
           "HMI_Interface_Overview".homeCodition[0].emOverviewCmPositionName[7] := WSTRING#'Spare';
           "HMI_Interface_Overview".homeCodition[0].emOverviewCmPositionName[8] := WSTRING#'Spare';
           "HMI_Interface_Overview".homeCodition[0].emOverviewCmPositionName[9] := WSTRING#'Spare';
           "HMI_Interface_Overview".homeCodition[0].emOverviewCmPositionName[10] := WSTRING#'Spare';
           "HMI_Interface_Overview".homeCodition[0].emOverviewCmPositionName[11] := WSTRING#'Spare';
           "HMI_Interface_Overview".homeCodition[0].emOverviewCmPositionName[12] := WSTRING#'Spare';
           "HMI_Interface_Overview".homeCodition[0].emOverviewCmPositionName[13] := WSTRING#'Spare';
           IF NOT #statLampControl THEN
               "HMI_Interface_Overview".homeCodition[0].emOverviewHomeLampOn[0] := "Unit1.Em0.HmiInterface".cmStacker1NgBoxLoadingUpDown.monitoring.inHomePos;
               "HMI_Interface_Overview".homeCodition[0].emOverviewHomeLampOn[1] := "Unit1.Em0.HmiInterface".cmStacker1NgBoxUnitMoverBwdFwd.monitoring.inHomePos;
               "HMI_Interface_Overview".homeCodition[0].emOverviewHomeLampOn[2] := "Unit1.Em0.HmiInterface".cmStacker1NgBoxClampLeftOpenClose.monitoring.inWorkPos;
               "HMI_Interface_Overview".homeCodition[0].emOverviewHomeLampOn[3] := "Unit1.Em0.HmiInterface".cmStacker1NgBoxClampRightOpenClose.monitoring.inWorkPos;
               "HMI_Interface_Overview".homeCodition[0].emOverviewHomeLampOn[4] := "Unit1.Em0.HmiInterface".cmStacker1NgBoxClampMoverOpenClose.monitoring.inWorkPos;
               "HMI_Interface_Overview".homeCodition[0].emOverviewHomeLampOn[5] := FALSE;
               "HMI_Interface_Overview".homeCodition[0].emOverviewHomeLampOn[6] := FALSE;
               "HMI_Interface_Overview".homeCodition[0].emOverviewHomeLampOn[7] := FALSE;
               "HMI_Interface_Overview".homeCodition[0].emOverviewHomeLampOn[8] := FALSE;
               "HMI_Interface_Overview".homeCodition[0].emOverviewHomeLampOn[9] := FALSE;
               "HMI_Interface_Overview".homeCodition[0].emOverviewHomeLampOn[10] := FALSE;
               "HMI_Interface_Overview".homeCodition[0].emOverviewHomeLampOn[11] := FALSE;
               "HMI_Interface_Overview".homeCodition[0].emOverviewHomeLampOn[12] := FALSE;
               "HMI_Interface_Overview".homeCodition[0].emOverviewHomeLampOn[13] := FALSE;
           END_IF;
       END_IF;

   END_REGION
END_REGION

REGION Network 31 (SCL): Em 1 Page Index Mapping
   REGION Page Index

       // Index 0
       IF "HMI_Interface_Overview".homeCodition[1].pageIndex = 0 THEN
           "HMI_Interface_Overview".homeCodition[1].emOverviewTitle := WSTRING#'Home Conidtion 0';
           "HMI_Interface_Overview".homeCodition[1].emOverviewCmName[0] := WSTRING#'Stacker 2 NG Box Loading';
           "HMI_Interface_Overview".homeCodition[1].emOverviewCmName[1] := WSTRING#'Stacker 2 NG Box Unit Mover';
           "HMI_Interface_Overview".homeCodition[1].emOverviewCmName[2] := WSTRING#'Stacker 2 NG Box Clamp Left';
           "HMI_Interface_Overview".homeCodition[1].emOverviewCmName[3] := WSTRING#'Stacker 2 NG Box Clamp Right';
           "HMI_Interface_Overview".homeCodition[1].emOverviewCmName[4] := WSTRING#'Stacker 2 NG Box Clamp Mover';
           "HMI_Interface_Overview".homeCodition[1].emOverviewCmName[5] := WSTRING#'Spare';
           "HMI_Interface_Overview".homeCodition[1].emOverviewCmName[6] := WSTRING#'Spare';
           "HMI_Interface_Overview".homeCodition[1].emOverviewCmName[7] := WSTRING#'Spare';
           "HMI_Interface_Overview".homeCodition[1].emOverviewCmName[8] := WSTRING#'Spare';
           "HMI_Interface_Overview".homeCodition[1].emOverviewCmName[9] := WSTRING#'Spare';
           "HMI_Interface_Overview".homeCodition[1].emOverviewCmName[10] := WSTRING#'Spare';
           "HMI_Interface_Overview".homeCodition[1].emOverviewCmName[11] := WSTRING#'Spare';
           "HMI_Interface_Overview".homeCodition[1].emOverviewCmName[12] := WSTRING#'Spare';
           "HMI_Interface_Overview".homeCodition[1].emOverviewCmName[13] := WSTRING#'Spare';
           "HMI_Interface_Overview".homeCodition[1].emOverviewCmPositionName[0] := WSTRING#'Up';
           "HMI_Interface_Overview".homeCodition[1].emOverviewCmPositionName[1] := WSTRING#'Backward';
           "HMI_Interface_Overview".homeCodition[1].emOverviewCmPositionName[2] := WSTRING#'Open';
           "HMI_Interface_Overview".homeCodition[1].emOverviewCmPositionName[3] := WSTRING#'Open';
           "HMI_Interface_Overview".homeCodition[1].emOverviewCmPositionName[4] := WSTRING#'Open';
           "HMI_Interface_Overview".homeCodition[1].emOverviewCmPositionName[5] := WSTRING#'Spare';
           "HMI_Interface_Overview".homeCodition[1].emOverviewCmPositionName[6] := WSTRING#'Spare';
           "HMI_Interface_Overview".homeCodition[1].emOverviewCmPositionName[7] := WSTRING#'Spare';
           "HMI_Interface_Overview".homeCodition[1].emOverviewCmPositionName[8] := WSTRING#'Spare';
           "HMI_Interface_Overview".homeCodition[1].emOverviewCmPositionName[9] := WSTRING#'Spare';
           "HMI_Interface_Overview".homeCodition[1].emOverviewCmPositionName[10] := WSTRING#'Spare';
           "HMI_Interface_Overview".homeCodition[1].emOverviewCmPositionName[11] := WSTRING#'Spare';
           "HMI_Interface_Overview".homeCodition[1].emOverviewCmPositionName[12] := WSTRING#'Spare';
           "HMI_Interface_Overview".homeCodition[1].emOverviewCmPositionName[13] := WSTRING#'Spare';
           IF NOT #statLampControl THEN
               "HMI_Interface_Overview".homeCodition[1].emOverviewHomeLampOn[0] := "Unit1.Em1.HmiInterface".cmStacker2NgBoxLoadingUpDown.monitoring.inHomePos;
               "HMI_Interface_Overview".homeCodition[1].emOverviewHomeLampOn[1] := "Unit1.Em1.HmiInterface".cmStacker2NgBoxUnitMoverBwdFwd.monitoring.inHomePos;
               "HMI_Interface_Overview".homeCodition[1].emOverviewHomeLampOn[2] := "Unit1.Em1.HmiInterface".cmStacker2NgBoxClampLeftOpenClose.monitoring.inHomePos;
               "HMI_Interface_Overview".homeCodition[1].emOverviewHomeLampOn[3] := "Unit1.Em1.HmiInterface".cmStacker2NgBoxClampRightOpenClose.monitoring.inHomePos;
               "HMI_Interface_Overview".homeCodition[1].emOverviewHomeLampOn[4] := "Unit1.Em1.HmiInterface".cmStacker2NgBoxClampMoverOpenClose.monitoring.inHomePos;
               "HMI_Interface_Overview".homeCodition[1].emOverviewHomeLampOn[5] := FALSE;
               "HMI_Interface_Overview".homeCodition[1].emOverviewHomeLampOn[6] := FALSE;
               "HMI_Interface_Overview".homeCodition[1].emOverviewHomeLampOn[7] := FALSE;
               "HMI_Interface_Overview".homeCodition[1].emOverviewHomeLampOn[8] := FALSE;
               "HMI_Interface_Overview".homeCodition[1].emOverviewHomeLampOn[9] := FALSE;
               "HMI_Interface_Overview".homeCodition[1].emOverviewHomeLampOn[10] := FALSE;
               "HMI_Interface_Overview".homeCodition[1].emOverviewHomeLampOn[11] := FALSE;
               "HMI_Interface_Overview".homeCodition[1].emOverviewHomeLampOn[12] := FALSE;
               "HMI_Interface_Overview".homeCodition[1].emOverviewHomeLampOn[13] := FALSE;
           END_IF;
       END_IF;

       // Index 1
       IF "HMI_Interface_Overview".homeCodition[1].pageIndex = 1 THEN
           "HMI_Interface_Overview".homeCodition[1].emOverviewTitle := WSTRING#'Home Conidtion 1';
           "HMI_Interface_Overview".homeCodition[1].emOverviewCmName[0] := WSTRING#'Stacker 2 NG Box Loading';
           "HMI_Interface_Overview".homeCodition[1].emOverviewCmName[1] := WSTRING#'Stacker 2 NG Box Unit Mover';
           "HMI_Interface_Overview".homeCodition[1].emOverviewCmName[2] := WSTRING#'Stacker 2 NG Box Clamp Left';
           "HMI_Interface_Overview".homeCodition[1].emOverviewCmName[3] := WSTRING#'Stacker 2 NG Box Clamp Right';
           "HMI_Interface_Overview".homeCodition[1].emOverviewCmName[4] := WSTRING#'Stacker 2 NG Box Clamp Mover';
           "HMI_Interface_Overview".homeCodition[1].emOverviewCmName[5] := WSTRING#'Spare';
           "HMI_Interface_Overview".homeCodition[1].emOverviewCmName[6] := WSTRING#'Spare';
           "HMI_Interface_Overview".homeCodition[1].emOverviewCmName[7] := WSTRING#'Spare';
           "HMI_Interface_Overview".homeCodition[1].emOverviewCmName[8] := WSTRING#'Spare';
           "HMI_Interface_Overview".homeCodition[1].emOverviewCmName[9] := WSTRING#'Spare';
           "HMI_Interface_Overview".homeCodition[1].emOverviewCmName[10] := WSTRING#'Spare';
           "HMI_Interface_Overview".homeCodition[1].emOverviewCmName[11] := WSTRING#'Spare';
           "HMI_Interface_Overview".homeCodition[1].emOverviewCmName[12] := WSTRING#'Spare';
           "HMI_Interface_Overview".homeCodition[1].emOverviewCmName[13] := WSTRING#'Spare';
           "HMI_Interface_Overview".homeCodition[1].emOverviewCmPositionName[0] := WSTRING#'Up';
           "HMI_Interface_Overview".homeCodition[1].emOverviewCmPositionName[1] := WSTRING#'Backward';
           "HMI_Interface_Overview".homeCodition[1].emOverviewCmPositionName[2] := WSTRING#'Close';
           "HMI_Interface_Overview".homeCodition[1].emOverviewCmPositionName[3] := WSTRING#'Close';
           "HMI_Interface_Overview".homeCodition[1].emOverviewCmPositionName[4] := WSTRING#'Close';
           "HMI_Interface_Overview".homeCodition[1].emOverviewCmPositionName[5] := WSTRING#'Spare';
           "HMI_Interface_Overview".homeCodition[1].emOverviewCmPositionName[6] := WSTRING#'Spare';
           "HMI_Interface_Overview".homeCodition[1].emOverviewCmPositionName[7] := WSTRING#'Spare';
           "HMI_Interface_Overview".homeCodition[1].emOverviewCmPositionName[8] := WSTRING#'Spare';
           "HMI_Interface_Overview".homeCodition[1].emOverviewCmPositionName[9] := WSTRING#'Spare';
           "HMI_Interface_Overview".homeCodition[1].emOverviewCmPositionName[10] := WSTRING#'Spare';
           "HMI_Interface_Overview".homeCodition[1].emOverviewCmPositionName[11] := WSTRING#'Spare';
           "HMI_Interface_Overview".homeCodition[1].emOverviewCmPositionName[12] := WSTRING#'Spare';
           "HMI_Interface_Overview".homeCodition[1].emOverviewCmPositionName[13] := WSTRING#'Spare';
           IF NOT #statLampControl THEN
               "HMI_Interface_Overview".homeCodition[1].emOverviewHomeLampOn[0] := "Unit1.Em1.HmiInterface".cmStacker2NgBoxLoadingUpDown.monitoring.inHomePos;
               "HMI_Interface_Overview".homeCodition[1].emOverviewHomeLampOn[1] := "Unit1.Em1.HmiInterface".cmStacker2NgBoxUnitMoverBwdFwd.monitoring.inHomePos;
               "HMI_Interface_Overview".homeCodition[1].emOverviewHomeLampOn[2] := "Unit1.Em1.HmiInterface".cmStacker2NgBoxClampLeftOpenClose.monitoring.inWorkPos;
               "HMI_Interface_Overview".homeCodition[1].emOverviewHomeLampOn[3] := "Unit1.Em1.HmiInterface".cmStacker2NgBoxClampRightOpenClose.monitoring.inWorkPos;
               "HMI_Interface_Overview".homeCodition[1].emOverviewHomeLampOn[4] := "Unit1.Em1.HmiInterface".cmStacker2NgBoxClampMoverOpenClose.monitoring.inWorkPos;
               "HMI_Interface_Overview".homeCodition[1].emOverviewHomeLampOn[5] := FALSE;
               "HMI_Interface_Overview".homeCodition[1].emOverviewHomeLampOn[6] := FALSE;
               "HMI_Interface_Overview".homeCodition[1].emOverviewHomeLampOn[7] := FALSE;
               "HMI_Interface_Overview".homeCodition[1].emOverviewHomeLampOn[8] := FALSE;
               "HMI_Interface_Overview".homeCodition[1].emOverviewHomeLampOn[9] := FALSE;
               "HMI_Interface_Overview".homeCodition[1].emOverviewHomeLampOn[10] := FALSE;
               "HMI_Interface_Overview".homeCodition[1].emOverviewHomeLampOn[11] := FALSE;
               "HMI_Interface_Overview".homeCodition[1].emOverviewHomeLampOn[12] := FALSE;
               "HMI_Interface_Overview".homeCodition[1].emOverviewHomeLampOn[13] := FALSE;
           END_IF;
       END_IF;

   END_REGION
END_REGION

REGION Network 32 (SCL): Em 2 Page Index Mapping
   REGION Page Index

       // Index 0
       IF "HMI_Interface_Overview".homeCodition[2].pageIndex = 0 THEN
           "HMI_Interface_Overview".homeCodition[2].emOverviewTitle := WSTRING#'P&P Left Home Condition 0';
           "HMI_Interface_Overview".homeCodition[2].emOverviewCmName[0] := WSTRING#'JR Out P&P Left X-Axis';
           "HMI_Interface_Overview".homeCodition[2].emOverviewCmName[1] := WSTRING#'JR Out P&P Left Z-Axis';
           "HMI_Interface_Overview".homeCodition[2].emOverviewCmName[2] := WSTRING#'JR Out P&P Left Clamp';
           "HMI_Interface_Overview".homeCodition[2].emOverviewCmName[3] := WSTRING#'JR Out P&P Left JR Detect';
           "HMI_Interface_Overview".homeCodition[2].emOverviewCmName[4] := WSTRING#'Spare';
           "HMI_Interface_Overview".homeCodition[2].emOverviewCmName[5] := WSTRING#'Spare';
           "HMI_Interface_Overview".homeCodition[2].emOverviewCmName[6] := WSTRING#'Spare';
           "HMI_Interface_Overview".homeCodition[2].emOverviewCmName[7] := WSTRING#'Spare';
           "HMI_Interface_Overview".homeCodition[2].emOverviewCmName[8] := WSTRING#'Spare';
           "HMI_Interface_Overview".homeCodition[2].emOverviewCmName[9] := WSTRING#'Spare';
           "HMI_Interface_Overview".homeCodition[2].emOverviewCmName[10] := WSTRING#'Spare';
           "HMI_Interface_Overview".homeCodition[2].emOverviewCmName[11] := WSTRING#'Spare';
           "HMI_Interface_Overview".homeCodition[2].emOverviewCmName[12] := WSTRING#'Spare';
           "HMI_Interface_Overview".homeCodition[2].emOverviewCmName[13] := WSTRING#'Spare';
           "HMI_Interface_Overview".homeCodition[2].emOverviewCmPositionName[0] := WSTRING#'Wait Position';
           "HMI_Interface_Overview".homeCodition[2].emOverviewCmPositionName[1] := WSTRING#'Wait Position';
           "HMI_Interface_Overview".homeCodition[2].emOverviewCmPositionName[2] := WSTRING#'Open';
           "HMI_Interface_Overview".homeCodition[2].emOverviewCmPositionName[3] := WSTRING#'Not Detect';
           "HMI_Interface_Overview".homeCodition[2].emOverviewCmPositionName[4] := WSTRING#'Spare';
           "HMI_Interface_Overview".homeCodition[2].emOverviewCmPositionName[5] := WSTRING#'Spare';
           "HMI_Interface_Overview".homeCodition[2].emOverviewCmPositionName[6] := WSTRING#'Spare';
           "HMI_Interface_Overview".homeCodition[2].emOverviewCmPositionName[7] := WSTRING#'Spare';
           "HMI_Interface_Overview".homeCodition[2].emOverviewCmPositionName[8] := WSTRING#'Spare';
           "HMI_Interface_Overview".homeCodition[2].emOverviewCmPositionName[9] := WSTRING#'Spare';
           "HMI_Interface_Overview".homeCodition[2].emOverviewCmPositionName[10] := WSTRING#'Spare';
           "HMI_Interface_Overview".homeCodition[2].emOverviewCmPositionName[11] := WSTRING#'Spare';
           "HMI_Interface_Overview".homeCodition[2].emOverviewCmPositionName[12] := WSTRING#'Spare';
           "HMI_Interface_Overview".homeCodition[2].emOverviewCmPositionName[13] := WSTRING#'Spare';
           IF NOT #statLampControl THEN
               "HMI_Interface_Overview".homeCodition[2].emOverviewHomeLampOn[0] := "Unit1.Em2.HmiInterface".cm.softcam.jrOutPnPLeftAxisX.pos00_wait.inPos;
               "HMI_Interface_Overview".homeCodition[2].emOverviewHomeLampOn[1] := "Unit1.Em2.HmiInterface".cm.softcam.jrOutPnPLeftAxisZ.pos01_stack1Load.inPos;
               "HMI_Interface_Overview".homeCodition[2].emOverviewHomeLampOn[2] := "Unit1.Em2.HmiInterface".cmJROutPnPLeftClampOpenClose.monitoring.inHomePos;
               "HMI_Interface_Overview".homeCodition[2].emOverviewHomeLampOn[3] := NOT "Unit1.Em2.HmiInterface".cmJROutPnPLeftJRDetect.monitoring.processValue;
               "HMI_Interface_Overview".homeCodition[2].emOverviewHomeLampOn[4] := FALSE;
               "HMI_Interface_Overview".homeCodition[2].emOverviewHomeLampOn[5] := FALSE;
               "HMI_Interface_Overview".homeCodition[2].emOverviewHomeLampOn[6] := FALSE;
               "HMI_Interface_Overview".homeCodition[2].emOverviewHomeLampOn[7] := FALSE;
               "HMI_Interface_Overview".homeCodition[2].emOverviewHomeLampOn[8] := FALSE;
               "HMI_Interface_Overview".homeCodition[2].emOverviewHomeLampOn[9] := FALSE;
               "HMI_Interface_Overview".homeCodition[2].emOverviewHomeLampOn[10] := FALSE;
               "HMI_Interface_Overview".homeCodition[2].emOverviewHomeLampOn[11] := FALSE;
               "HMI_Interface_Overview".homeCodition[2].emOverviewHomeLampOn[12] := FALSE;
               "HMI_Interface_Overview".homeCodition[2].emOverviewHomeLampOn[13] := FALSE;
           END_IF;
       END_IF;

       // Index 1
       IF "HMI_Interface_Overview".homeCodition[2].pageIndex = 1 THEN
           "HMI_Interface_Overview".homeCodition[2].emOverviewTitle := WSTRING#'P&P Left Home Condition 1';
           "HMI_Interface_Overview".homeCodition[2].emOverviewCmName[0] := WSTRING#'JR Out P&P Left X-Axis';
           "HMI_Interface_Overview".homeCodition[2].emOverviewCmName[1] := WSTRING#'JR Out P&P Left Z-Axis';
           "HMI_Interface_Overview".homeCodition[2].emOverviewCmName[2] := WSTRING#'JR Out P&P Left Clamp';
           "HMI_Interface_Overview".homeCodition[2].emOverviewCmName[3] := WSTRING#'JR Out P&P Left JR Detect';
           "HMI_Interface_Overview".homeCodition[2].emOverviewCmName[4] := WSTRING#'Spare';
           "HMI_Interface_Overview".homeCodition[2].emOverviewCmName[5] := WSTRING#'Spare';
           "HMI_Interface_Overview".homeCodition[2].emOverviewCmName[6] := WSTRING#'Spare';
           "HMI_Interface_Overview".homeCodition[2].emOverviewCmName[7] := WSTRING#'Spare';
           "HMI_Interface_Overview".homeCodition[2].emOverviewCmName[8] := WSTRING#'Spare';
           "HMI_Interface_Overview".homeCodition[2].emOverviewCmName[9] := WSTRING#'Spare';
           "HMI_Interface_Overview".homeCodition[2].emOverviewCmName[10] := WSTRING#'Spare';
           "HMI_Interface_Overview".homeCodition[2].emOverviewCmName[11] := WSTRING#'Spare';
           "HMI_Interface_Overview".homeCodition[2].emOverviewCmName[12] := WSTRING#'Spare';
           "HMI_Interface_Overview".homeCodition[2].emOverviewCmName[13] := WSTRING#'Spare';
           "HMI_Interface_Overview".homeCodition[2].emOverviewCmPositionName[0] := WSTRING#'Wait Position';
           "HMI_Interface_Overview".homeCodition[2].emOverviewCmPositionName[1] := WSTRING#'Wait Position';
           "HMI_Interface_Overview".homeCodition[2].emOverviewCmPositionName[2] := WSTRING#'Close';
           "HMI_Interface_Overview".homeCodition[2].emOverviewCmPositionName[3] := WSTRING#'Detect';
           "HMI_Interface_Overview".homeCodition[2].emOverviewCmPositionName[4] := WSTRING#'Spare';
           "HMI_Interface_Overview".homeCodition[2].emOverviewCmPositionName[5] := WSTRING#'Spare';
           "HMI_Interface_Overview".homeCodition[2].emOverviewCmPositionName[6] := WSTRING#'Spare';
           "HMI_Interface_Overview".homeCodition[2].emOverviewCmPositionName[7] := WSTRING#'Spare';
           "HMI_Interface_Overview".homeCodition[2].emOverviewCmPositionName[8] := WSTRING#'Spare';
           "HMI_Interface_Overview".homeCodition[2].emOverviewCmPositionName[9] := WSTRING#'Spare';
           "HMI_Interface_Overview".homeCodition[2].emOverviewCmPositionName[10] := WSTRING#'Spare';
           "HMI_Interface_Overview".homeCodition[2].emOverviewCmPositionName[11] := WSTRING#'Spare';
           "HMI_Interface_Overview".homeCodition[2].emOverviewCmPositionName[12] := WSTRING#'Spare';
           "HMI_Interface_Overview".homeCodition[2].emOverviewCmPositionName[13] := WSTRING#'Spare';
           IF NOT #statLampControl THEN
               "HMI_Interface_Overview".homeCodition[2].emOverviewHomeLampOn[0] := "Unit1.Em2.HmiInterface".cm.softcam.jrOutPnPLeftAxisX.pos00_wait.inPos;
               "HMI_Interface_Overview".homeCodition[2].emOverviewHomeLampOn[1] := "Unit1.Em2.HmiInterface".cm.softcam.jrOutPnPLeftAxisZ.pos00_wait.inPos;
               "HMI_Interface_Overview".homeCodition[2].emOverviewHomeLampOn[2] := "Unit1.Em2.HmiInterface".cmJROutPnPLeftClampOpenClose.monitoring.inWorkPos;
               "HMI_Interface_Overview".homeCodition[2].emOverviewHomeLampOn[3] := "Unit1.Em2.HmiInterface".cmJROutPnPLeftJRDetect.monitoring.processValue;
               "HMI_Interface_Overview".homeCodition[2].emOverviewHomeLampOn[4] := FALSE;
               "HMI_Interface_Overview".homeCodition[2].emOverviewHomeLampOn[5] := FALSE;
               "HMI_Interface_Overview".homeCodition[2].emOverviewHomeLampOn[6] := FALSE;
               "HMI_Interface_Overview".homeCodition[2].emOverviewHomeLampOn[7] := FALSE;
               "HMI_Interface_Overview".homeCodition[2].emOverviewHomeLampOn[8] := FALSE;
               "HMI_Interface_Overview".homeCodition[2].emOverviewHomeLampOn[9] := FALSE;
               "HMI_Interface_Overview".homeCodition[2].emOverviewHomeLampOn[10] := FALSE;
               "HMI_Interface_Overview".homeCodition[2].emOverviewHomeLampOn[11] := FALSE;
               "HMI_Interface_Overview".homeCodition[2].emOverviewHomeLampOn[12] := FALSE;
               "HMI_Interface_Overview".homeCodition[2].emOverviewHomeLampOn[13] := FALSE;
           END_IF;
       END_IF;

       // Index 2
       IF "HMI_Interface_Overview".homeCodition[2].pageIndex = 2 THEN
           "HMI_Interface_Overview".homeCodition[2].emOverviewTitle := WSTRING#'P&P Right Home Condition 0';
           "HMI_Interface_Overview".homeCodition[2].emOverviewCmName[0] := WSTRING#'JR Out P&P Right X-Axis';
           "HMI_Interface_Overview".homeCodition[2].emOverviewCmName[1] := WSTRING#'JR Out P&P Right Z-Axis';
           "HMI_Interface_Overview".homeCodition[2].emOverviewCmName[2] := WSTRING#'JR Out P&P Right Clamp';
           "HMI_Interface_Overview".homeCodition[2].emOverviewCmName[3] := WSTRING#'JR Out P&P Right JR Detect';
           "HMI_Interface_Overview".homeCodition[2].emOverviewCmName[4] := WSTRING#'Spare';
           "HMI_Interface_Overview".homeCodition[2].emOverviewCmName[5] := WSTRING#'Spare';
           "HMI_Interface_Overview".homeCodition[2].emOverviewCmName[6] := WSTRING#'Spare';
           "HMI_Interface_Overview".homeCodition[2].emOverviewCmName[7] := WSTRING#'Spare';
           "HMI_Interface_Overview".homeCodition[2].emOverviewCmName[8] := WSTRING#'Spare';
           "HMI_Interface_Overview".homeCodition[2].emOverviewCmName[9] := WSTRING#'Spare';
           "HMI_Interface_Overview".homeCodition[2].emOverviewCmName[10] := WSTRING#'Spare';
           "HMI_Interface_Overview".homeCodition[2].emOverviewCmName[11] := WSTRING#'Spare';
           "HMI_Interface_Overview".homeCodition[2].emOverviewCmName[12] := WSTRING#'Spare';
           "HMI_Interface_Overview".homeCodition[2].emOverviewCmName[13] := WSTRING#'Spare';
           "HMI_Interface_Overview".homeCodition[2].emOverviewCmPositionName[0] := WSTRING#'Wait Position';
           "HMI_Interface_Overview".homeCodition[2].emOverviewCmPositionName[1] := WSTRING#'Wait Position';
           "HMI_Interface_Overview".homeCodition[2].emOverviewCmPositionName[2] := WSTRING#'Open';
           "HMI_Interface_Overview".homeCodition[2].emOverviewCmPositionName[3] := WSTRING#'Not Detect';
           "HMI_Interface_Overview".homeCodition[2].emOverviewCmPositionName[4] := WSTRING#'Spare';
           "HMI_Interface_Overview".homeCodition[2].emOverviewCmPositionName[5] := WSTRING#'Spare';
           "HMI_Interface_Overview".homeCodition[2].emOverviewCmPositionName[6] := WSTRING#'Spare';
           "HMI_Interface_Overview".homeCodition[2].emOverviewCmPositionName[7] := WSTRING#'Spare';
           "HMI_Interface_Overview".homeCodition[2].emOverviewCmPositionName[8] := WSTRING#'Spare';
           "HMI_Interface_Overview".homeCodition[2].emOverviewCmPositionName[9] := WSTRING#'Spare';
           "HMI_Interface_Overview".homeCodition[2].emOverviewCmPositionName[10] := WSTRING#'Spare';
           "HMI_Interface_Overview".homeCodition[2].emOverviewCmPositionName[11] := WSTRING#'Spare';
           "HMI_Interface_Overview".homeCodition[2].emOverviewCmPositionName[12] := WSTRING#'Spare';
           "HMI_Interface_Overview".homeCodition[2].emOverviewCmPositionName[13] := WSTRING#'Spare';
           IF NOT #statLampControl THEN
               "HMI_Interface_Overview".homeCodition[2].emOverviewHomeLampOn[0] := "Unit1.Em2.HmiInterface".cm.softcam.jrOutPnPLeftAxisX.pos00_wait.inPos;
               "HMI_Interface_Overview".homeCodition[2].emOverviewHomeLampOn[1] := "Unit1.Em2.HmiInterface".cm.softcam.jrOutPnPLeftAxisZ.pos00_wait.inPos;
               "HMI_Interface_Overview".homeCodition[2].emOverviewHomeLampOn[2] := "Unit1.Em2.HmiInterface".cmJROutPnPRightClampOpenClose.monitoring.inHomePos;
               "HMI_Interface_Overview".homeCodition[2].emOverviewHomeLampOn[3] := NOT "Unit1.Em2.HmiInterface".cmJROutPnPRightJRDetect.monitoring.processValue;
               "HMI_Interface_Overview".homeCodition[2].emOverviewHomeLampOn[4] := FALSE;
               "HMI_Interface_Overview".homeCodition[2].emOverviewHomeLampOn[5] := FALSE;
               "HMI_Interface_Overview".homeCodition[2].emOverviewHomeLampOn[6] := FALSE;
               "HMI_Interface_Overview".homeCodition[2].emOverviewHomeLampOn[7] := FALSE;
               "HMI_Interface_Overview".homeCodition[2].emOverviewHomeLampOn[8] := FALSE;
               "HMI_Interface_Overview".homeCodition[2].emOverviewHomeLampOn[9] := FALSE;
               "HMI_Interface_Overview".homeCodition[2].emOverviewHomeLampOn[10] := FALSE;
               "HMI_Interface_Overview".homeCodition[2].emOverviewHomeLampOn[11] := FALSE;
               "HMI_Interface_Overview".homeCodition[2].emOverviewHomeLampOn[12] := FALSE;
               "HMI_Interface_Overview".homeCodition[2].emOverviewHomeLampOn[13] := FALSE;
           END_IF;
       END_IF;

       // Index 3
       IF "HMI_Interface_Overview".homeCodition[2].pageIndex = 3 THEN
           "HMI_Interface_Overview".homeCodition[2].emOverviewTitle := WSTRING#'P&P Right Home Condition 1';
           "HMI_Interface_Overview".homeCodition[2].emOverviewCmName[0] := WSTRING#'JR Out P&P Right X-Axis';
           "HMI_Interface_Overview".homeCodition[2].emOverviewCmName[1] := WSTRING#'JR Out P&P Right Z-Axis';
           "HMI_Interface_Overview".homeCodition[2].emOverviewCmName[2] := WSTRING#'JR Out P&P Right Clamp';
           "HMI_Interface_Overview".homeCodition[2].emOverviewCmName[3] := WSTRING#'JR Out P&P Right JR Detect';
           "HMI_Interface_Overview".homeCodition[2].emOverviewCmName[4] := WSTRING#'Spare';
           "HMI_Interface_Overview".homeCodition[2].emOverviewCmName[5] := WSTRING#'Spare';
           "HMI_Interface_Overview".homeCodition[2].emOverviewCmName[6] := WSTRING#'Spare';
           "HMI_Interface_Overview".homeCodition[2].emOverviewCmName[7] := WSTRING#'Spare';
           "HMI_Interface_Overview".homeCodition[2].emOverviewCmName[8] := WSTRING#'Spare';
           "HMI_Interface_Overview".homeCodition[2].emOverviewCmName[9] := WSTRING#'Spare';
           "HMI_Interface_Overview".homeCodition[2].emOverviewCmName[10] := WSTRING#'Spare';
           "HMI_Interface_Overview".homeCodition[2].emOverviewCmName[11] := WSTRING#'Spare';
           "HMI_Interface_Overview".homeCodition[2].emOverviewCmName[12] := WSTRING#'Spare';
           "HMI_Interface_Overview".homeCodition[2].emOverviewCmName[13] := WSTRING#'Spare';
           "HMI_Interface_Overview".homeCodition[2].emOverviewCmPositionName[0] := WSTRING#'Wait Position';
           "HMI_Interface_Overview".homeCodition[2].emOverviewCmPositionName[1] := WSTRING#'Wait Position';
           "HMI_Interface_Overview".homeCodition[2].emOverviewCmPositionName[2] := WSTRING#'Close';
           "HMI_Interface_Overview".homeCodition[2].emOverviewCmPositionName[3] := WSTRING#'Detect';
           "HMI_Interface_Overview".homeCodition[2].emOverviewCmPositionName[4] := WSTRING#'Spare';
           "HMI_Interface_Overview".homeCodition[2].emOverviewCmPositionName[5] := WSTRING#'Spare';
           "HMI_Interface_Overview".homeCodition[2].emOverviewCmPositionName[6] := WSTRING#'Spare';
           "HMI_Interface_Overview".homeCodition[2].emOverviewCmPositionName[7] := WSTRING#'Spare';
           "HMI_Interface_Overview".homeCodition[2].emOverviewCmPositionName[8] := WSTRING#'Spare';
           "HMI_Interface_Overview".homeCodition[2].emOverviewCmPositionName[9] := WSTRING#'Spare';
           "HMI_Interface_Overview".homeCodition[2].emOverviewCmPositionName[10] := WSTRING#'Spare';
           "HMI_Interface_Overview".homeCodition[2].emOverviewCmPositionName[11] := WSTRING#'Spare';
           "HMI_Interface_Overview".homeCodition[2].emOverviewCmPositionName[12] := WSTRING#'Spare';
           "HMI_Interface_Overview".homeCodition[2].emOverviewCmPositionName[13] := WSTRING#'Spare';
           IF NOT #statLampControl THEN
               "HMI_Interface_Overview".homeCodition[2].emOverviewHomeLampOn[0] := "Unit1.Em2.HmiInterface".cm.softcam.jrOutPnPLeftAxisX.pos00_wait.inPos;
               "HMI_Interface_Overview".homeCodition[2].emOverviewHomeLampOn[1] := "Unit1.Em2.HmiInterface".cm.softcam.jrOutPnPLeftAxisZ.pos00_wait.inPos;
               "HMI_Interface_Overview".homeCodition[2].emOverviewHomeLampOn[2] := "Unit1.Em2.HmiInterface".cmJROutPnPRightClampOpenClose.monitoring.inWorkPos;
               "HMI_Interface_Overview".homeCodition[2].emOverviewHomeLampOn[3] := "Unit1.Em2.HmiInterface".cmJROutPnPRightJRDetect.monitoring.processValue;
               "HMI_Interface_Overview".homeCodition[2].emOverviewHomeLampOn[4] := FALSE;
               "HMI_Interface_Overview".homeCodition[2].emOverviewHomeLampOn[5] := FALSE;
               "HMI_Interface_Overview".homeCodition[2].emOverviewHomeLampOn[6] := FALSE;
               "HMI_Interface_Overview".homeCodition[2].emOverviewHomeLampOn[7] := FALSE;
               "HMI_Interface_Overview".homeCodition[2].emOverviewHomeLampOn[8] := FALSE;
               "HMI_Interface_Overview".homeCodition[2].emOverviewHomeLampOn[9] := FALSE;
               "HMI_Interface_Overview".homeCodition[2].emOverviewHomeLampOn[10] := FALSE;
               "HMI_Interface_Overview".homeCodition[2].emOverviewHomeLampOn[11] := FALSE;
               "HMI_Interface_Overview".homeCodition[2].emOverviewHomeLampOn[12] := FALSE;
               "HMI_Interface_Overview".homeCodition[2].emOverviewHomeLampOn[13] := FALSE;
           END_IF;
       END_IF;

   END_REGION
END_REGION

REGION Network 33 (SCL): Em 3 Page Index Mapping
   REGION Page Index

       // Index 0
       IF "HMI_Interface_Overview".homeCodition[3].pageIndex = 0 THEN
           "HMI_Interface_Overview".homeCodition[3].emOverviewTitle := WSTRING#'Loading Home Condition 0';
           "HMI_Interface_Overview".homeCodition[3].emOverviewCmName[0] := WSTRING#'Top Tape Loading';
           "HMI_Interface_Overview".homeCodition[3].emOverviewCmName[1] := WSTRING#'Top Tape Loading Clamp';
           "HMI_Interface_Overview".homeCodition[3].emOverviewCmName[2] := WSTRING#'Top Tape Cutter';
           "HMI_Interface_Overview".homeCodition[3].emOverviewCmName[3] := WSTRING#'Top Tape Cutter Clamp';
           "HMI_Interface_Overview".homeCodition[3].emOverviewCmName[4] := WSTRING#'Top Tape Tension';
           "HMI_Interface_Overview".homeCodition[3].emOverviewCmName[5] := WSTRING#'Spare';
           "HMI_Interface_Overview".homeCodition[3].emOverviewCmName[6] := WSTRING#'Spare';
           "HMI_Interface_Overview".homeCodition[3].emOverviewCmName[7] := WSTRING#'Spare';
           "HMI_Interface_Overview".homeCodition[3].emOverviewCmName[8] := WSTRING#'Spare';
           "HMI_Interface_Overview".homeCodition[3].emOverviewCmName[9] := WSTRING#'Spare';
           "HMI_Interface_Overview".homeCodition[3].emOverviewCmName[10] := WSTRING#'Spare';
           "HMI_Interface_Overview".homeCodition[3].emOverviewCmName[11] := WSTRING#'Spare';
           "HMI_Interface_Overview".homeCodition[3].emOverviewCmName[12] := WSTRING#'Spare';
           "HMI_Interface_Overview".homeCodition[3].emOverviewCmName[13] := WSTRING#'Spare';
           "HMI_Interface_Overview".homeCodition[3].emOverviewCmPositionName[0] := WSTRING#'Backward';
           "HMI_Interface_Overview".homeCodition[3].emOverviewCmPositionName[1] := WSTRING#'Open';
           "HMI_Interface_Overview".homeCodition[3].emOverviewCmPositionName[2] := WSTRING#'Up';
           "HMI_Interface_Overview".homeCodition[3].emOverviewCmPositionName[3] := WSTRING#'Down';
           "HMI_Interface_Overview".homeCodition[3].emOverviewCmPositionName[4] := WSTRING#'Backward';
           "HMI_Interface_Overview".homeCodition[3].emOverviewCmPositionName[5] := WSTRING#'Spare';
           "HMI_Interface_Overview".homeCodition[3].emOverviewCmPositionName[6] := WSTRING#'Spare';
           "HMI_Interface_Overview".homeCodition[3].emOverviewCmPositionName[7] := WSTRING#'Spare';
           "HMI_Interface_Overview".homeCodition[3].emOverviewCmPositionName[8] := WSTRING#'Spare';
           "HMI_Interface_Overview".homeCodition[3].emOverviewCmPositionName[9] := WSTRING#'Spare';
           "HMI_Interface_Overview".homeCodition[3].emOverviewCmPositionName[10] := WSTRING#'Spare';
           "HMI_Interface_Overview".homeCodition[3].emOverviewCmPositionName[11] := WSTRING#'Spare';
           "HMI_Interface_Overview".homeCodition[3].emOverviewCmPositionName[12] := WSTRING#'Spare';
           "HMI_Interface_Overview".homeCodition[3].emOverviewCmPositionName[13] := WSTRING#'Spare';
           IF NOT #statLampControl THEN
               "HMI_Interface_Overview".homeCodition[3].emOverviewHomeLampOn[0] := "Unit1.Em3.HmiInterface".cmTopTapeLoadingBwdFwd.monitoring.inHomePos;
               "HMI_Interface_Overview".homeCodition[3].emOverviewHomeLampOn[1] := "Unit1.Em3.HmiInterface".cmTopTapeLoadingClampOpenClose.monitoring.inHomePos;
               "HMI_Interface_Overview".homeCodition[3].emOverviewHomeLampOn[2] := "Unit1.Em3.HmiInterface".cmTopTapeCutterUpDown.monitoring.inHomePos;
               "HMI_Interface_Overview".homeCodition[3].emOverviewHomeLampOn[3] := "Unit1.Em3.HmiInterface".cmTopTapeCutterClampUpDown.monitoring.inWorkPos;
               "HMI_Interface_Overview".homeCodition[3].emOverviewHomeLampOn[4] := "Unit1.Em3.HmiInterface".cmTopTapeTensionBwdFwd.monitoring.inHomePos;
               "HMI_Interface_Overview".homeCodition[3].emOverviewHomeLampOn[5] := FALSE;
               "HMI_Interface_Overview".homeCodition[3].emOverviewHomeLampOn[6] := FALSE;
               "HMI_Interface_Overview".homeCodition[3].emOverviewHomeLampOn[7] := FALSE;
               "HMI_Interface_Overview".homeCodition[3].emOverviewHomeLampOn[8] := FALSE;
               "HMI_Interface_Overview".homeCodition[3].emOverviewHomeLampOn[9] := FALSE;
               "HMI_Interface_Overview".homeCodition[3].emOverviewHomeLampOn[10] := FALSE;
               "HMI_Interface_Overview".homeCodition[3].emOverviewHomeLampOn[11] := FALSE;
               "HMI_Interface_Overview".homeCodition[3].emOverviewHomeLampOn[12] := FALSE;
               "HMI_Interface_Overview".homeCodition[3].emOverviewHomeLampOn[13] := FALSE;
           END_IF;
       END_IF;

       // Index 1
       IF "HMI_Interface_Overview".homeCodition[3].pageIndex = 1 THEN
           "HMI_Interface_Overview".homeCodition[3].emOverviewTitle := WSTRING#'Loading Home Condition 1';
           "HMI_Interface_Overview".homeCodition[3].emOverviewCmName[0] := WSTRING#'Top Tape Loading';
           "HMI_Interface_Overview".homeCodition[3].emOverviewCmName[1] := WSTRING#'Top Tape Loading Clamp';
           "HMI_Interface_Overview".homeCodition[3].emOverviewCmName[2] := WSTRING#'Top Tape Cutter';
           "HMI_Interface_Overview".homeCodition[3].emOverviewCmName[3] := WSTRING#'Top Tape Cutter Clamp';
           "HMI_Interface_Overview".homeCodition[3].emOverviewCmName[4] := WSTRING#'Top Tape Tension';
           "HMI_Interface_Overview".homeCodition[3].emOverviewCmName[5] := WSTRING#'Spare';
           "HMI_Interface_Overview".homeCodition[3].emOverviewCmName[6] := WSTRING#'Spare';
           "HMI_Interface_Overview".homeCodition[3].emOverviewCmName[7] := WSTRING#'Spare';
           "HMI_Interface_Overview".homeCodition[3].emOverviewCmName[8] := WSTRING#'Spare';
           "HMI_Interface_Overview".homeCodition[3].emOverviewCmName[9] := WSTRING#'Spare';
           "HMI_Interface_Overview".homeCodition[3].emOverviewCmName[10] := WSTRING#'Spare';
           "HMI_Interface_Overview".homeCodition[3].emOverviewCmName[11] := WSTRING#'Spare';
           "HMI_Interface_Overview".homeCodition[3].emOverviewCmName[12] := WSTRING#'Spare';
           "HMI_Interface_Overview".homeCodition[3].emOverviewCmName[13] := WSTRING#'Spare';
           "HMI_Interface_Overview".homeCodition[3].emOverviewCmPositionName[0] := WSTRING#'Backward';
           "HMI_Interface_Overview".homeCodition[3].emOverviewCmPositionName[1] := WSTRING#'Close';
           "HMI_Interface_Overview".homeCodition[3].emOverviewCmPositionName[2] := WSTRING#'Up';
           "HMI_Interface_Overview".homeCodition[3].emOverviewCmPositionName[3] := WSTRING#'Down';
           "HMI_Interface_Overview".homeCodition[3].emOverviewCmPositionName[4] := WSTRING#'Backward';
           "HMI_Interface_Overview".homeCodition[3].emOverviewCmPositionName[5] := WSTRING#'Spare';
           "HMI_Interface_Overview".homeCodition[3].emOverviewCmPositionName[6] := WSTRING#'Spare';
           "HMI_Interface_Overview".homeCodition[3].emOverviewCmPositionName[7] := WSTRING#'Spare';
           "HMI_Interface_Overview".homeCodition[3].emOverviewCmPositionName[8] := WSTRING#'Spare';
           "HMI_Interface_Overview".homeCodition[3].emOverviewCmPositionName[9] := WSTRING#'Spare';
           "HMI_Interface_Overview".homeCodition[3].emOverviewCmPositionName[10] := WSTRING#'Spare';
           "HMI_Interface_Overview".homeCodition[3].emOverviewCmPositionName[11] := WSTRING#'Spare';
           "HMI_Interface_Overview".homeCodition[3].emOverviewCmPositionName[12] := WSTRING#'Spare';
           "HMI_Interface_Overview".homeCodition[3].emOverviewCmPositionName[13] := WSTRING#'Spare';
           IF NOT #statLampControl THEN
               "HMI_Interface_Overview".homeCodition[3].emOverviewHomeLampOn[0] := "Unit1.Em3.HmiInterface".cmTopTapeLoadingBwdFwd.monitoring.inHomePos;
               "HMI_Interface_Overview".homeCodition[3].emOverviewHomeLampOn[1] := "Unit1.Em3.HmiInterface".cmTopTapeLoadingClampOpenClose.monitoring.inWorkPos;
               "HMI_Interface_Overview".homeCodition[3].emOverviewHomeLampOn[2] := "Unit1.Em3.HmiInterface".cmTopTapeCutterUpDown.monitoring.inHomePos;
               "HMI_Interface_Overview".homeCodition[3].emOverviewHomeLampOn[3] := "Unit1.Em3.HmiInterface".cmTopTapeCutterClampUpDown.monitoring.inWorkPos;
               "HMI_Interface_Overview".homeCodition[3].emOverviewHomeLampOn[4] := "Unit1.Em3.HmiInterface".cmTopTapeTensionBwdFwd.monitoring.inHomePos;
               "HMI_Interface_Overview".homeCodition[3].emOverviewHomeLampOn[5] := FALSE;
               "HMI_Interface_Overview".homeCodition[3].emOverviewHomeLampOn[6] := FALSE;
               "HMI_Interface_Overview".homeCodition[3].emOverviewHomeLampOn[7] := FALSE;
               "HMI_Interface_Overview".homeCodition[3].emOverviewHomeLampOn[8] := FALSE;
               "HMI_Interface_Overview".homeCodition[3].emOverviewHomeLampOn[9] := FALSE;
               "HMI_Interface_Overview".homeCodition[3].emOverviewHomeLampOn[10] := FALSE;
               "HMI_Interface_Overview".homeCodition[3].emOverviewHomeLampOn[11] := FALSE;
               "HMI_Interface_Overview".homeCodition[3].emOverviewHomeLampOn[12] := FALSE;
               "HMI_Interface_Overview".homeCodition[3].emOverviewHomeLampOn[13] := FALSE;
           END_IF;
       END_IF;

       // Index 2
       IF "HMI_Interface_Overview".homeCodition[3].pageIndex = 2 THEN
           "HMI_Interface_Overview".homeCodition[3].emOverviewTitle := WSTRING#'Attachment Home Condition 0';
           "HMI_Interface_Overview".homeCodition[3].emOverviewCmName[0] := WSTRING#'Top Tape X-Axis';
           "HMI_Interface_Overview".homeCodition[3].emOverviewCmName[1] := WSTRING#'Top Tape Attachment';
           "HMI_Interface_Overview".homeCodition[3].emOverviewCmName[2] := WSTRING#'Top Tape Attachment Vacuum';
           "HMI_Interface_Overview".homeCodition[3].emOverviewCmName[3] := WSTRING#'Spare';
           "HMI_Interface_Overview".homeCodition[3].emOverviewCmName[4] := WSTRING#'Spare';
           "HMI_Interface_Overview".homeCodition[3].emOverviewCmName[5] := WSTRING#'Spare';
           "HMI_Interface_Overview".homeCodition[3].emOverviewCmName[6] := WSTRING#'Spare';
           "HMI_Interface_Overview".homeCodition[3].emOverviewCmName[7] := WSTRING#'Spare';
           "HMI_Interface_Overview".homeCodition[3].emOverviewCmName[8] := WSTRING#'Spare';
           "HMI_Interface_Overview".homeCodition[3].emOverviewCmName[9] := WSTRING#'Spare';
           "HMI_Interface_Overview".homeCodition[3].emOverviewCmName[10] := WSTRING#'Spare';
           "HMI_Interface_Overview".homeCodition[3].emOverviewCmName[11] := WSTRING#'Spare';
           "HMI_Interface_Overview".homeCodition[3].emOverviewCmName[12] := WSTRING#'Spare';
           "HMI_Interface_Overview".homeCodition[3].emOverviewCmName[13] := WSTRING#'Spare';
           "HMI_Interface_Overview".homeCodition[3].emOverviewCmPositionName[0] := WSTRING#'Wait Position';
           "HMI_Interface_Overview".homeCodition[3].emOverviewCmPositionName[1] := WSTRING#'Up';
           "HMI_Interface_Overview".homeCodition[3].emOverviewCmPositionName[2] := WSTRING#'Off';
           "HMI_Interface_Overview".homeCodition[3].emOverviewCmPositionName[3] := WSTRING#'Spare';
           "HMI_Interface_Overview".homeCodition[3].emOverviewCmPositionName[4] := WSTRING#'Spare';
           "HMI_Interface_Overview".homeCodition[3].emOverviewCmPositionName[5] := WSTRING#'Spare';
           "HMI_Interface_Overview".homeCodition[3].emOverviewCmPositionName[6] := WSTRING#'Spare';
           "HMI_Interface_Overview".homeCodition[3].emOverviewCmPositionName[7] := WSTRING#'Spare';
           "HMI_Interface_Overview".homeCodition[3].emOverviewCmPositionName[8] := WSTRING#'Spare';
           "HMI_Interface_Overview".homeCodition[3].emOverviewCmPositionName[9] := WSTRING#'Spare';
           "HMI_Interface_Overview".homeCodition[3].emOverviewCmPositionName[10] := WSTRING#'Spare';
           "HMI_Interface_Overview".homeCodition[3].emOverviewCmPositionName[11] := WSTRING#'Spare';
           "HMI_Interface_Overview".homeCodition[3].emOverviewCmPositionName[12] := WSTRING#'Spare';
           "HMI_Interface_Overview".homeCodition[3].emOverviewCmPositionName[13] := WSTRING#'Spare';
           IF NOT #statLampControl THEN
               "HMI_Interface_Overview".homeCodition[3].emOverviewHomeLampOn[0] := "Unit1.Em3.HmiInterface".cm.softcam.topTapeAxisX.pos00_wait.inPos;
               "HMI_Interface_Overview".homeCodition[3].emOverviewHomeLampOn[1] := "Unit1.Em3.HmiInterface".cmTopTapeAttachmentUpDown.monitoring.inHomePos;
               "HMI_Interface_Overview".homeCodition[3].emOverviewHomeLampOn[2] := "Unit1.Em3.HmiInterface".cmTopTapeAttachmentVaccumOffOn.monitoring.inHomePos;
               "HMI_Interface_Overview".homeCodition[3].emOverviewHomeLampOn[3] := FALSE;
               "HMI_Interface_Overview".homeCodition[3].emOverviewHomeLampOn[4] := FALSE;
               "HMI_Interface_Overview".homeCodition[3].emOverviewHomeLampOn[5] := FALSE;
               "HMI_Interface_Overview".homeCodition[3].emOverviewHomeLampOn[6] := FALSE;
               "HMI_Interface_Overview".homeCodition[3].emOverviewHomeLampOn[7] := FALSE;
               "HMI_Interface_Overview".homeCodition[3].emOverviewHomeLampOn[8] := FALSE;
               "HMI_Interface_Overview".homeCodition[3].emOverviewHomeLampOn[9] := FALSE;
               "HMI_Interface_Overview".homeCodition[3].emOverviewHomeLampOn[10] := FALSE;
               "HMI_Interface_Overview".homeCodition[3].emOverviewHomeLampOn[11] := FALSE;
               "HMI_Interface_Overview".homeCodition[3].emOverviewHomeLampOn[12] := FALSE;
               "HMI_Interface_Overview".homeCodition[3].emOverviewHomeLampOn[13] := FALSE;
           END_IF;
       END_IF;

